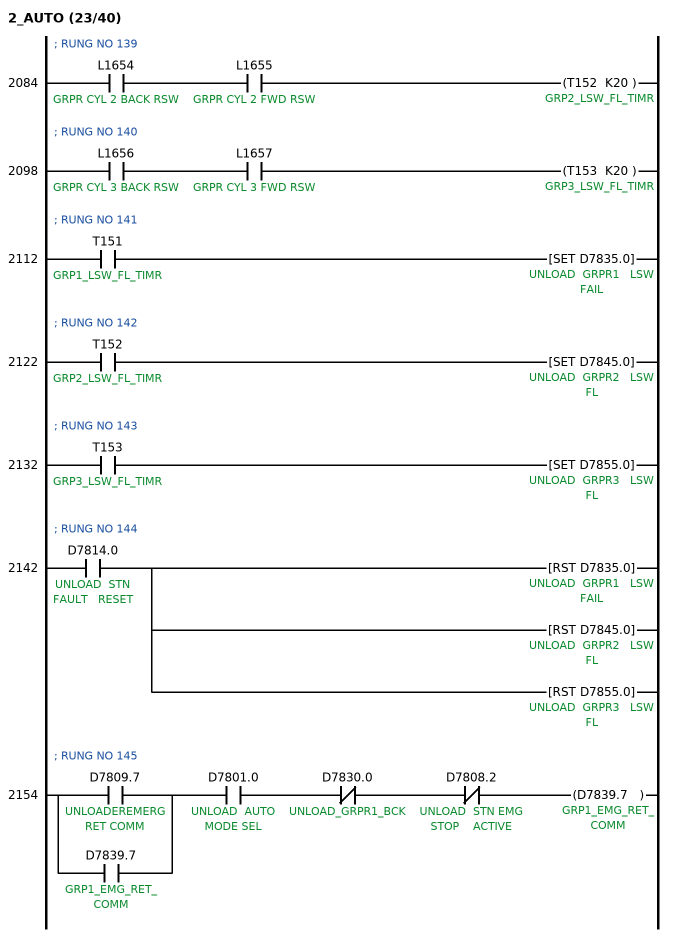
; RUNG NO 139
2084  LD      L1654  ; GRPR CYL 2 BACK RSW
      AND     L1655  ; GRPR CYL 2 FWD RSW
      OUT     T152 K20  ; GRP2_LSW_FL_TIMR
; RUNG NO 140
2098  LD      L1656  ; GRPR CYL 3 BACK RSW
      AND     L1657  ; GRPR CYL 3 FWD RSW
      OUT     T153 K20  ; GRP3_LSW_FL_TIMR
; RUNG NO 141
2112  LD      T151  ; GRP1_LSW_FL_TIMR
      SET     D7835.0  ; UNLOAD  GRPR1   LSW FAIL
; RUNG NO 142
2122  LD      T152  ; GRP2_LSW_FL_TIMR
      SET     D7845.0  ; UNLOAD  GRPR2   LSW FL
; RUNG NO 143
2132  LD      T153  ; GRP3_LSW_FL_TIMR
      SET     D7855.0  ; UNLOAD  GRPR3   LSW FL
; RUNG NO 144
2142  LD      D7814.0  ; UNLOAD  STN     FAULT   RESET
      RST     D7835.0  ; UNLOAD  GRPR1   LSW FAIL
      RST     D7845.0  ; UNLOAD  GRPR2   LSW FL
      RST     D7855.0  ; UNLOAD  GRPR3   LSW FL
; RUNG NO 145
2154  LD      D7809.7  ; UNLOADEREMERG   RET COMM
      OR      D7839.7  ; GRP1_EMG_RET_COMM
      AND     D7801.0  ; UNLOAD  AUTO    MODE SEL
      ANI     D7830.0  ; UNLOAD_GRPR1_BCK
      ANI     D7808.2  ; UNLOAD  STN EMG STOP    ACTIVE
      OUT     D7839.7  ; GRP1_EMG_RET_COMM
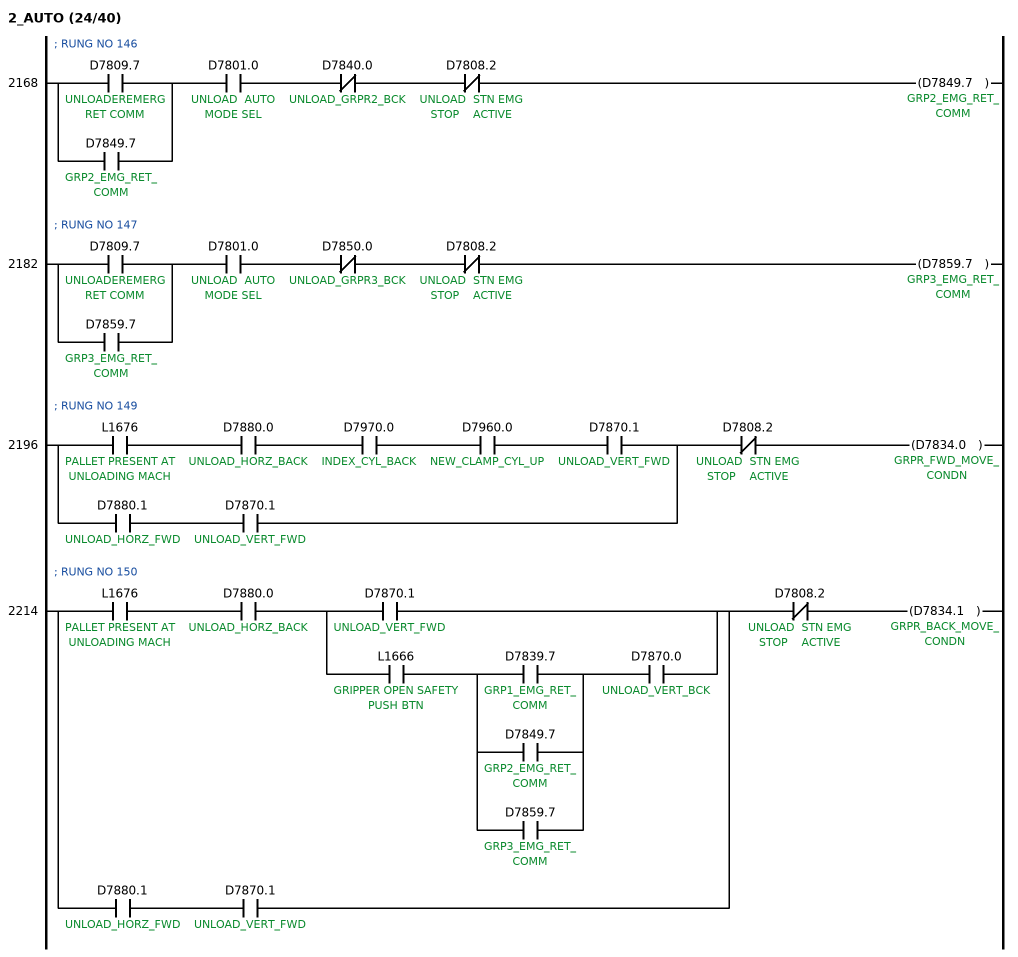
; RUNG NO 146
2168  LD      D7809.7  ; UNLOADEREMERG   RET COMM
      OR      D7849.7  ; GRP2_EMG_RET_COMM
      AND     D7801.0  ; UNLOAD  AUTO    MODE SEL
      ANI     D7840.0  ; UNLOAD_GRPR2_BCK
      ANI     D7808.2  ; UNLOAD  STN EMG STOP    ACTIVE
      OUT     D7849.7  ; GRP2_EMG_RET_COMM
; RUNG NO 147
2182  LD      D7809.7  ; UNLOADEREMERG   RET COMM
      OR      D7859.7  ; GRP3_EMG_RET_COMM
      AND     D7801.0  ; UNLOAD  AUTO    MODE SEL
      ANI     D7850.0  ; UNLOAD_GRPR3_BCK
      ANI     D7808.2  ; UNLOAD  STN EMG STOP    ACTIVE
      OUT     D7859.7  ; GRP3_EMG_RET_COMM
; RUNG NO 149
2196  LD      L1676  ; PALLET PRESENT AT UNLOADING MACH
      AND     D7880.0  ; UNLOAD_HORZ_BACK
      AND     D7970.0  ; INDEX_CYL_BACK
      AND     D7960.0  ; NEW_CLAMP_CYL_UP
      AND     D7870.1  ; UNLOAD_VERT_FWD
      LD      D7880.1  ; UNLOAD_HORZ_FWD
      AND     D7870.1  ; UNLOAD_VERT_FWD
      ORB
      ANI     D7808.2  ; UNLOAD  STN EMG STOP    ACTIVE
      OUT     D7834.0  ; GRPR_FWD_MOVE_CONDN
; RUNG NO 150
2214  LD      L1676  ; PALLET PRESENT AT UNLOADING MACH
      AND     D7880.0  ; UNLOAD_HORZ_BACK
      LD      D7870.1  ; UNLOAD_VERT_FWD
      LD      L1666  ; GRIPPER OPEN SAFETY PUSH BTN
      LD      D7839.7  ; GRP1_EMG_RET_COMM
      OR      D7849.7  ; GRP2_EMG_RET_COMM
      OR      D7859.7  ; GRP3_EMG_RET_COMM
      ANB
      AND     D7870.0  ; UNLOAD_VERT_BCK
      ORB
      ANB
      LD      D7880.1  ; UNLOAD_HORZ_FWD
      AND     D7870.1  ; UNLOAD_VERT_FWD
      ORB
      ANI     D7808.2  ; UNLOAD  STN EMG STOP    ACTIVE
      OUT     D7834.1  ; GRPR_BACK_MOVE_CONDN
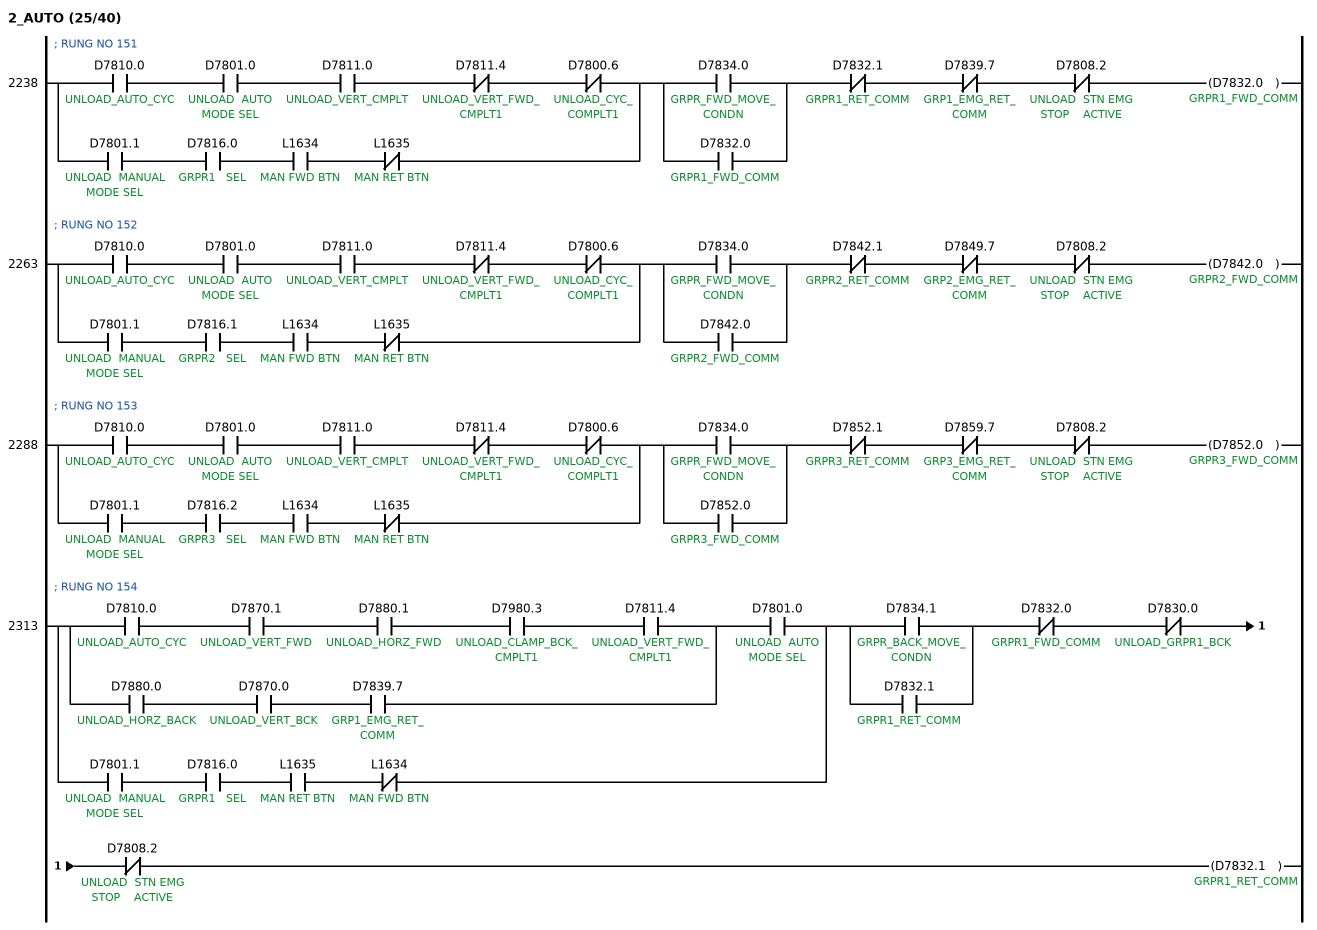
; RUNG NO 151
2238  LD      D7810.0  ; UNLOAD_AUTO_CYC
      AND     D7801.0  ; UNLOAD  AUTO    MODE SEL
      AND     D7811.0  ; UNLOAD_VERT_CMPLT
      ANI     D7811.4  ; UNLOAD_VERT_FWD_CMPLT1
      ANI     D7800.6  ; UNLOAD_CYC_COMPLT1
      LD      D7801.1  ; UNLOAD  MANUAL  MODE SEL
      AND     D7816.0  ; GRPR1   SEL
      AND     L1634  ; MAN FWD BTN
      ANI     L1635  ; MAN RET BTN
      ORB
      LD      D7834.0  ; GRPR_FWD_MOVE_CONDN
      OR      D7832.0  ; GRPR1_FWD_COMM
      ANB
      ANI     D7832.1  ; GRPR1_RET_COMM
      ANI     D7839.7  ; GRP1_EMG_RET_COMM
      ANI     D7808.2  ; UNLOAD  STN EMG STOP    ACTIVE
      OUT     D7832.0  ; GRPR1_FWD_COMM
; RUNG NO 152
2263  LD      D7810.0  ; UNLOAD_AUTO_CYC
      AND     D7801.0  ; UNLOAD  AUTO    MODE SEL
      AND     D7811.0  ; UNLOAD_VERT_CMPLT
      ANI     D7811.4  ; UNLOAD_VERT_FWD_CMPLT1
      ANI     D7800.6  ; UNLOAD_CYC_COMPLT1
      LD      D7801.1  ; UNLOAD  MANUAL  MODE SEL
      AND     D7816.1  ; GRPR2   SEL
      AND     L1634  ; MAN FWD BTN
      ANI     L1635  ; MAN RET BTN
      ORB
      LD      D7834.0  ; GRPR_FWD_MOVE_CONDN
      OR      D7842.0  ; GRPR2_FWD_COMM
      ANB
      ANI     D7842.1  ; GRPR2_RET_COMM
      ANI     D7849.7  ; GRP2_EMG_RET_COMM
      ANI     D7808.2  ; UNLOAD  STN EMG STOP    ACTIVE
      OUT     D7842.0  ; GRPR2_FWD_COMM
; RUNG NO 153
2288  LD      D7810.0  ; UNLOAD_AUTO_CYC
      AND     D7801.0  ; UNLOAD  AUTO    MODE SEL
      AND     D7811.0  ; UNLOAD_VERT_CMPLT
      ANI     D7811.4  ; UNLOAD_VERT_FWD_CMPLT1
      ANI     D7800.6  ; UNLOAD_CYC_COMPLT1
      LD      D7801.1  ; UNLOAD  MANUAL  MODE SEL
      AND     D7816.2  ; GRPR3   SEL
      AND     L1634  ; MAN FWD BTN
      ANI     L1635  ; MAN RET BTN
      ORB
      LD      D7834.0  ; GRPR_FWD_MOVE_CONDN
      OR      D7852.0  ; GRPR3_FWD_COMM
      ANB
      ANI     D7852.1  ; GRPR3_RET_COMM
      ANI     D7859.7  ; GRP3_EMG_RET_COMM
      ANI     D7808.2  ; UNLOAD  STN EMG STOP    ACTIVE
      OUT     D7852.0  ; GRPR3_FWD_COMM
; RUNG NO 154
2313  LD      D7810.0  ; UNLOAD_AUTO_CYC
      AND     D7870.1  ; UNLOAD_VERT_FWD
      AND     D7880.1  ; UNLOAD_HORZ_FWD
      AND     D7980.3  ; UNLOAD_CLAMP_BCK_CMPLT1
      AND     D7811.4  ; UNLOAD_VERT_FWD_CMPLT1
      LD      D7880.0  ; UNLOAD_HORZ_BACK
      AND     D7870.0  ; UNLOAD_VERT_BCK
      AND     D7839.7  ; GRP1_EMG_RET_COMM
      ORB
      AND     D7801.0  ; UNLOAD  AUTO    MODE SEL
      LD      D7801.1  ; UNLOAD  MANUAL  MODE SEL
      AND     D7816.0  ; GRPR1   SEL
      AND     L1635  ; MAN RET BTN
      ANI     L1634  ; MAN FWD BTN
      ORB
      LD      D7834.1  ; GRPR_BACK_MOVE_CONDN
      OR      D7832.1  ; GRPR1_RET_COMM
      ANB
      ANI     D7832.0  ; GRPR1_FWD_COMM
      ANI     D7830.0  ; UNLOAD_GRPR1_BCK
      ANI     D7808.2  ; UNLOAD  STN EMG STOP    ACTIVE
      OUT     D7832.1  ; GRPR1_RET_COMM
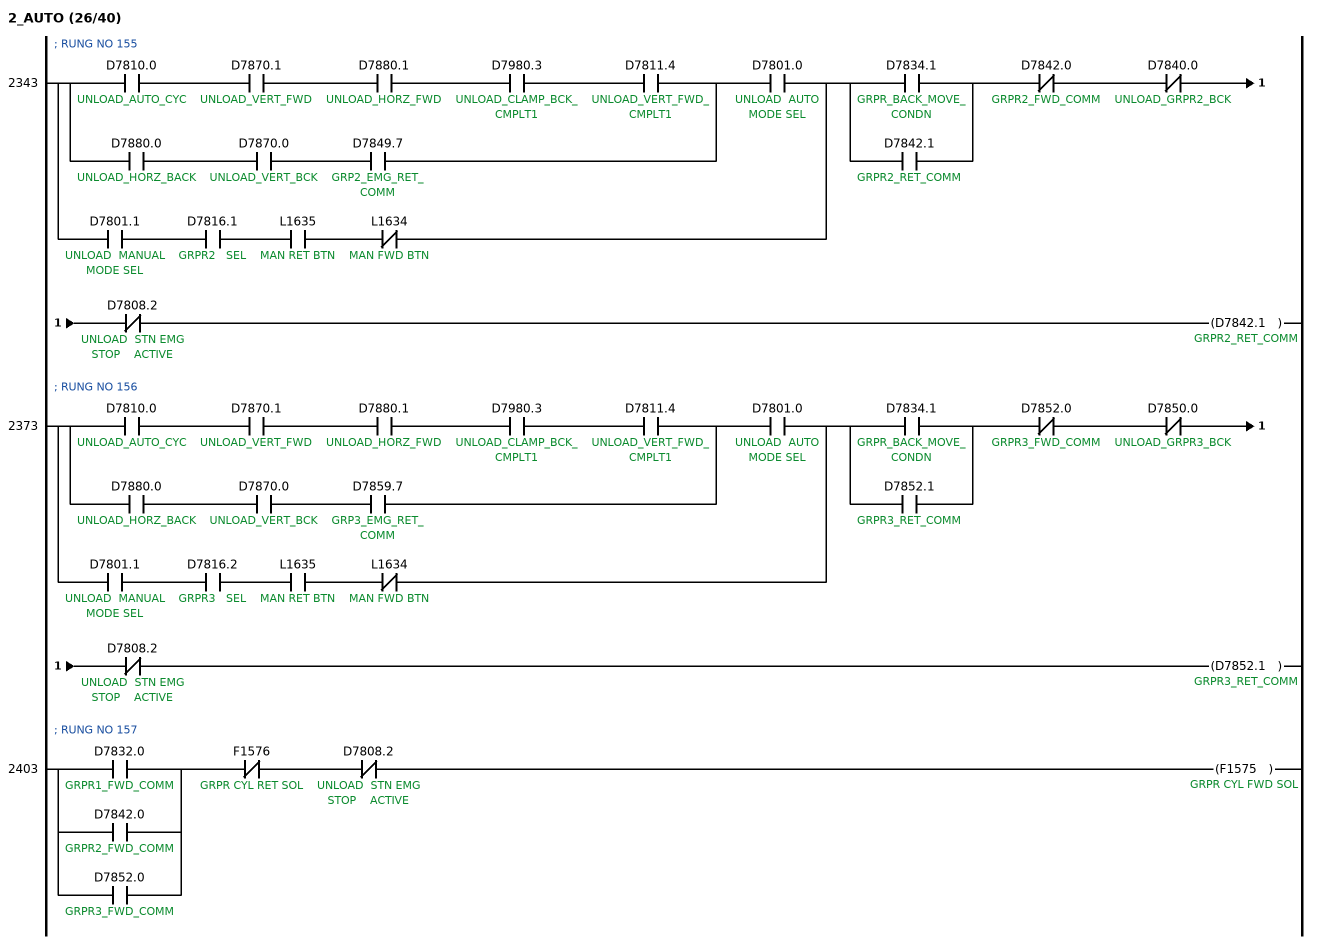
; RUNG NO 155
2343  LD      D7810.0  ; UNLOAD_AUTO_CYC
      AND     D7870.1  ; UNLOAD_VERT_FWD
      AND     D7880.1  ; UNLOAD_HORZ_FWD
      AND     D7980.3  ; UNLOAD_CLAMP_BCK_CMPLT1
      AND     D7811.4  ; UNLOAD_VERT_FWD_CMPLT1
      LD      D7880.0  ; UNLOAD_HORZ_BACK
      AND     D7870.0  ; UNLOAD_VERT_BCK
      AND     D7849.7  ; GRP2_EMG_RET_COMM
      ORB
      AND     D7801.0  ; UNLOAD  AUTO    MODE SEL
      LD      D7801.1  ; UNLOAD  MANUAL  MODE SEL
      AND     D7816.1  ; GRPR2   SEL
      AND     L1635  ; MAN RET BTN
      ANI     L1634  ; MAN FWD BTN
      ORB
      LD      D7834.1  ; GRPR_BACK_MOVE_CONDN
      OR      D7842.1  ; GRPR2_RET_COMM
      ANB
      ANI     D7842.0  ; GRPR2_FWD_COMM
      ANI     D7840.0  ; UNLOAD_GRPR2_BCK
      ANI     D7808.2  ; UNLOAD  STN EMG STOP    ACTIVE
      OUT     D7842.1  ; GRPR2_RET_COMM
; RUNG NO 156
2373  LD      D7810.0  ; UNLOAD_AUTO_CYC
      AND     D7870.1  ; UNLOAD_VERT_FWD
      AND     D7880.1  ; UNLOAD_HORZ_FWD
      AND     D7980.3  ; UNLOAD_CLAMP_BCK_CMPLT1
      AND     D7811.4  ; UNLOAD_VERT_FWD_CMPLT1
      LD      D7880.0  ; UNLOAD_HORZ_BACK
      AND     D7870.0  ; UNLOAD_VERT_BCK
      AND     D7859.7  ; GRP3_EMG_RET_COMM
      ORB
      AND     D7801.0  ; UNLOAD  AUTO    MODE SEL
      LD      D7801.1  ; UNLOAD  MANUAL  MODE SEL
      AND     D7816.2  ; GRPR3   SEL
      AND     L1635  ; MAN RET BTN
      ANI     L1634  ; MAN FWD BTN
      ORB
      LD      D7834.1  ; GRPR_BACK_MOVE_CONDN
      OR      D7852.1  ; GRPR3_RET_COMM
      ANB
      ANI     D7852.0  ; GRPR3_FWD_COMM
      ANI     D7850.0  ; UNLOAD_GRPR3_BCK
      ANI     D7808.2  ; UNLOAD  STN EMG STOP    ACTIVE
      OUT     D7852.1  ; GRPR3_RET_COMM
; RUNG NO 157
2403  LD      D7832.0  ; GRPR1_FWD_COMM
      OR      D7842.0  ; GRPR2_FWD_COMM
      OR      D7852.0  ; GRPR3_FWD_COMM
      ANI     F1576  ; GRPR CYL RET SOL
      ANI     D7808.2  ; UNLOAD  STN EMG STOP    ACTIVE
      OUT     F1575  ; GRPR CYL FWD SOL
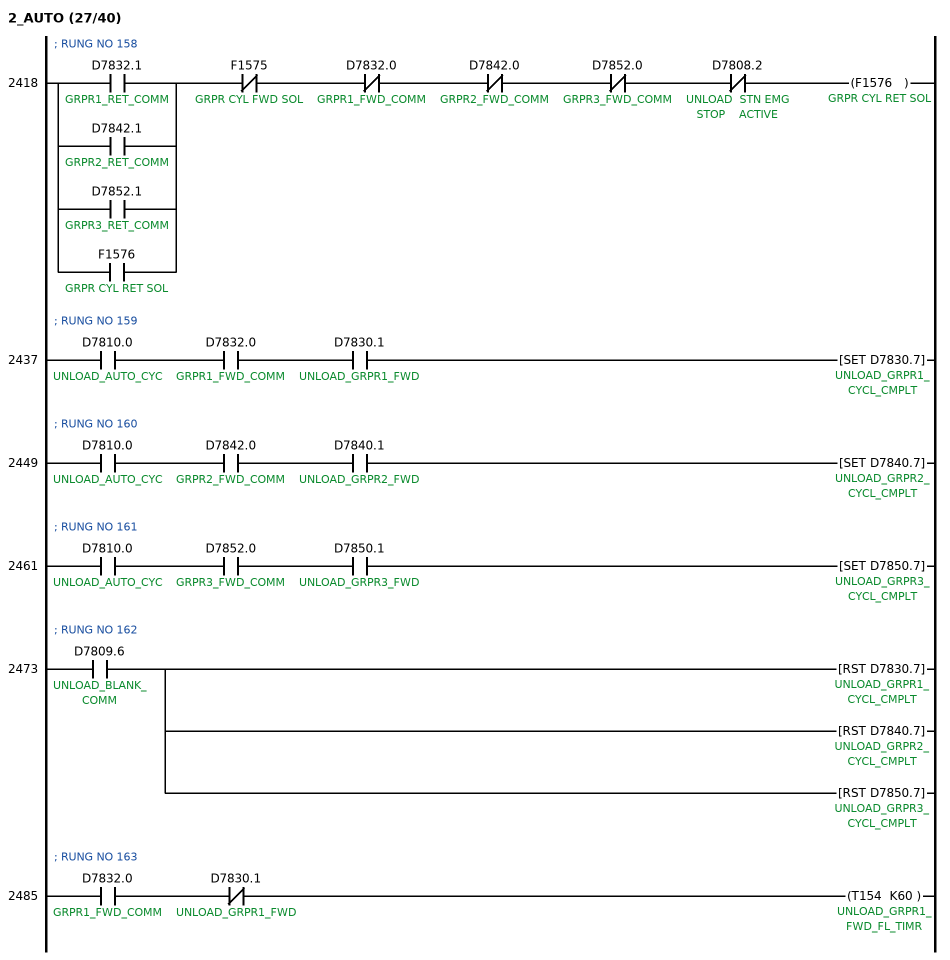
; RUNG NO 158
2418  LD      D7832.1  ; GRPR1_RET_COMM
      OR      D7842.1  ; GRPR2_RET_COMM
      OR      D7852.1  ; GRPR3_RET_COMM
      OR      F1576  ; GRPR CYL RET SOL
      ANI     F1575  ; GRPR CYL FWD SOL
      ANI     D7832.0  ; GRPR1_FWD_COMM
      ANI     D7842.0  ; GRPR2_FWD_COMM
      ANI     D7852.0  ; GRPR3_FWD_COMM
      ANI     D7808.2  ; UNLOAD  STN EMG STOP    ACTIVE
      OUT     F1576  ; GRPR CYL RET SOL
; RUNG NO 159
2437  LD      D7810.0  ; UNLOAD_AUTO_CYC
      AND     D7832.0  ; GRPR1_FWD_COMM
      AND     D7830.1  ; UNLOAD_GRPR1_FWD
      SET     D7830.7  ; UNLOAD_GRPR1_CYCL_CMPLT
; RUNG NO 160
2449  LD      D7810.0  ; UNLOAD_AUTO_CYC
      AND     D7842.0  ; GRPR2_FWD_COMM
      AND     D7840.1  ; UNLOAD_GRPR2_FWD
      SET     D7840.7  ; UNLOAD_GRPR2_CYCL_CMPLT
; RUNG NO 161
2461  LD      D7810.0  ; UNLOAD_AUTO_CYC
      AND     D7852.0  ; GRPR3_FWD_COMM
      AND     D7850.1  ; UNLOAD_GRPR3_FWD
      SET     D7850.7  ; UNLOAD_GRPR3_CYCL_CMPLT
; RUNG NO 162
2473  LD      D7809.6  ; UNLOAD_BLANK_COMM
      RST     D7830.7  ; UNLOAD_GRPR1_CYCL_CMPLT
      RST     D7840.7  ; UNLOAD_GRPR2_CYCL_CMPLT
      RST     D7850.7  ; UNLOAD_GRPR3_CYCL_CMPLT
; RUNG NO 163
2485  LD      D7832.0  ; GRPR1_FWD_COMM
      ANI     D7830.1  ; UNLOAD_GRPR1_FWD
      OUT     T154 K60  ; UNLOAD_GRPR1_FWD_FL_TIMR
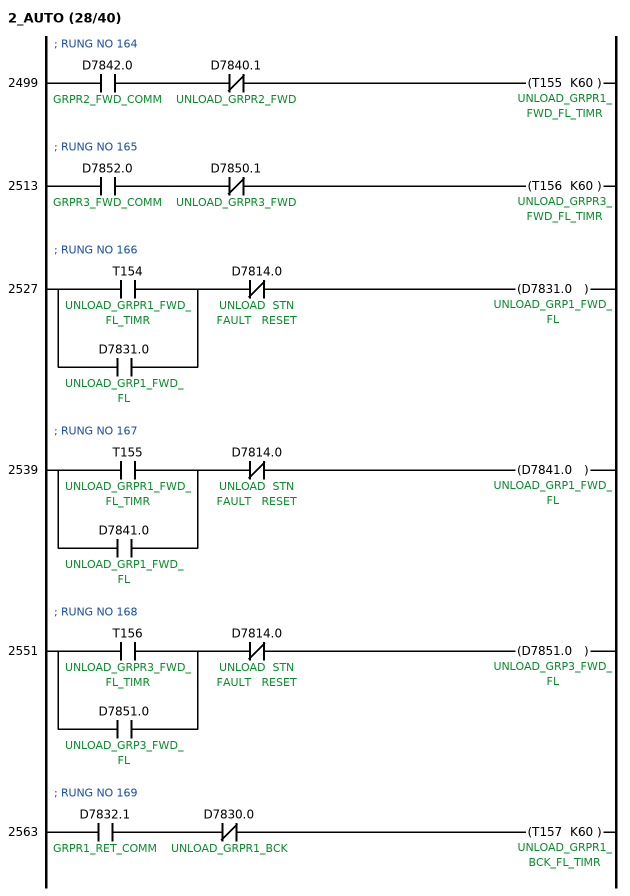
; RUNG NO 164
2499  LD      D7842.0  ; GRPR2_FWD_COMM
      ANI     D7840.1  ; UNLOAD_GRPR2_FWD
      OUT     T155 K60  ; UNLOAD_GRPR1_FWD_FL_TIMR
; RUNG NO 165
2513  LD      D7852.0  ; GRPR3_FWD_COMM
      ANI     D7850.1  ; UNLOAD_GRPR3_FWD
      OUT     T156 K60  ; UNLOAD_GRPR3_FWD_FL_TIMR
; RUNG NO 166
2527  LD      T154  ; UNLOAD_GRPR1_FWD_FL_TIMR
      OR      D7831.0  ; UNLOAD_GRP1_FWD_FL
      ANI     D7814.0  ; UNLOAD  STN     FAULT   RESET
      OUT     D7831.0  ; UNLOAD_GRP1_FWD_FL
; RUNG NO 167
2539  LD      T155  ; UNLOAD_GRPR1_FWD_FL_TIMR
      OR      D7841.0  ; UNLOAD_GRP1_FWD_FL
      ANI     D7814.0  ; UNLOAD  STN     FAULT   RESET
      OUT     D7841.0  ; UNLOAD_GRP1_FWD_FL
; RUNG NO 168
2551  LD      T156  ; UNLOAD_GRPR3_FWD_FL_TIMR
      OR      D7851.0  ; UNLOAD_GRP3_FWD_FL
      ANI     D7814.0  ; UNLOAD  STN     FAULT   RESET
      OUT     D7851.0  ; UNLOAD_GRP3_FWD_FL
; RUNG NO 169
2563  LD      D7832.1  ; GRPR1_RET_COMM
      ANI     D7830.0  ; UNLOAD_GRPR1_BCK
      OUT     T157 K60  ; UNLOAD_GRPR1_BCK_FL_TIMR
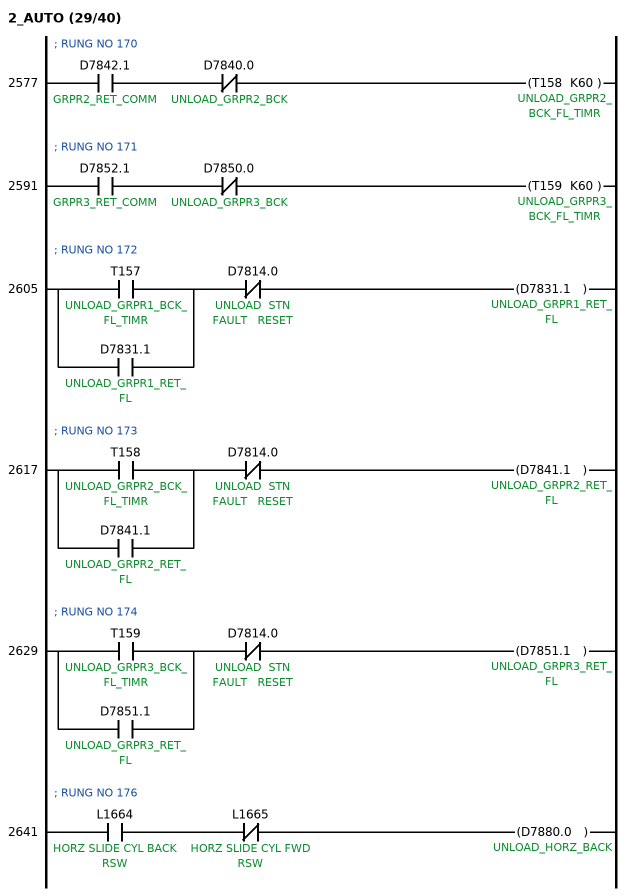
; RUNG NO 170
2577  LD      D7842.1  ; GRPR2_RET_COMM
      ANI     D7840.0  ; UNLOAD_GRPR2_BCK
      OUT     T158 K60  ; UNLOAD_GRPR2_BCK_FL_TIMR
; RUNG NO 171
2591  LD      D7852.1  ; GRPR3_RET_COMM
      ANI     D7850.0  ; UNLOAD_GRPR3_BCK
      OUT     T159 K60  ; UNLOAD_GRPR3_BCK_FL_TIMR
; RUNG NO 172
2605  LD      T157  ; UNLOAD_GRPR1_BCK_FL_TIMR
      OR      D7831.1  ; UNLOAD_GRPR1_RET_FL
      ANI     D7814.0  ; UNLOAD  STN     FAULT   RESET
      OUT     D7831.1  ; UNLOAD_GRPR1_RET_FL
; RUNG NO 173
2617  LD      T158  ; UNLOAD_GRPR2_BCK_FL_TIMR
      OR      D7841.1  ; UNLOAD_GRPR2_RET_FL
      ANI     D7814.0  ; UNLOAD  STN     FAULT   RESET
      OUT     D7841.1  ; UNLOAD_GRPR2_RET_FL
; RUNG NO 174
2629  LD      T159  ; UNLOAD_GRPR3_BCK_FL_TIMR
      OR      D7851.1  ; UNLOAD_GRPR3_RET_FL
      ANI     D7814.0  ; UNLOAD  STN     FAULT   RESET
      OUT     D7851.1  ; UNLOAD_GRPR3_RET_FL
; RUNG NO 176
2641  LD      L1664  ; HORZ SLIDE CYL BACK RSW
      ANI     L1665  ; HORZ SLIDE CYL FWD RSW
      OUT     D7880.0  ; UNLOAD_HORZ_BACK
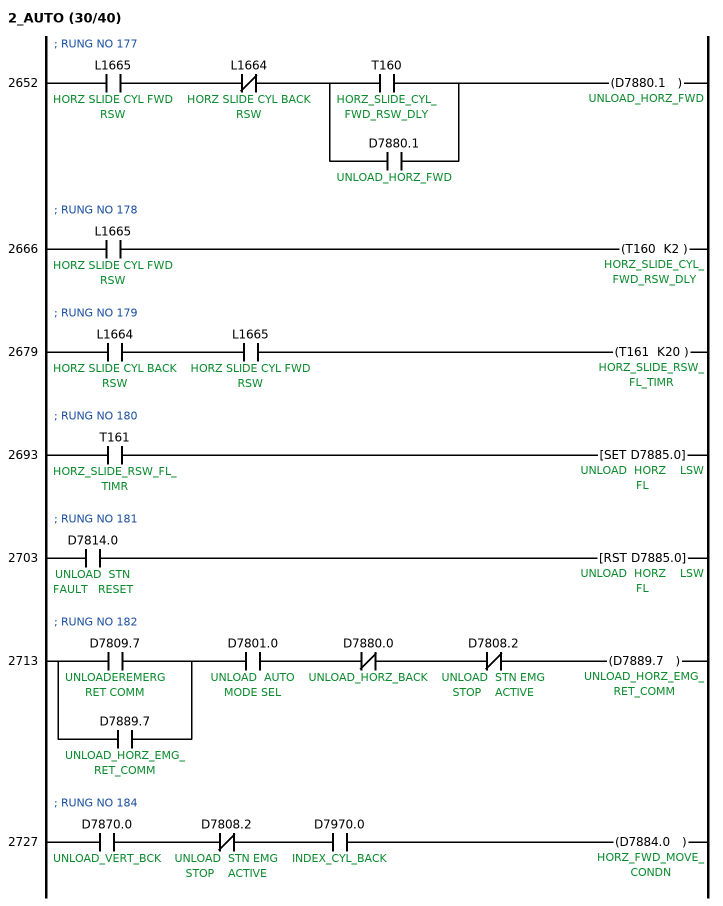
; RUNG NO 177
2652  LD      L1665  ; HORZ SLIDE CYL FWD RSW
      ANI     L1664  ; HORZ SLIDE CYL BACK RSW
      LD      T160  ; HORZ_SLIDE_CYL_FWD_RSW_DLY
      OR      D7880.1  ; UNLOAD_HORZ_FWD
      ANB
      OUT     D7880.1  ; UNLOAD_HORZ_FWD
; RUNG NO 178
2666  LD      L1665  ; HORZ SLIDE CYL FWD RSW
      OUT     T160 K2  ; HORZ_SLIDE_CYL_FWD_RSW_DLY
; RUNG NO 179
2679  LD      L1664  ; HORZ SLIDE CYL BACK RSW
      AND     L1665  ; HORZ SLIDE CYL FWD RSW
      OUT     T161 K20  ; HORZ_SLIDE_RSW_FL_TIMR
; RUNG NO 180
2693  LD      T161  ; HORZ_SLIDE_RSW_FL_TIMR
      SET     D7885.0  ; UNLOAD  HORZ    LSW FL
; RUNG NO 181
2703  LD      D7814.0  ; UNLOAD  STN     FAULT   RESET
      RST     D7885.0  ; UNLOAD  HORZ    LSW FL
; RUNG NO 182
2713  LD      D7809.7  ; UNLOADEREMERG   RET COMM
      OR      D7889.7  ; UNLOAD_HORZ_EMG_RET_COMM
      AND     D7801.0  ; UNLOAD  AUTO    MODE SEL
      ANI     D7880.0  ; UNLOAD_HORZ_BACK
      ANI     D7808.2  ; UNLOAD  STN EMG STOP    ACTIVE
      OUT     D7889.7  ; UNLOAD_HORZ_EMG_RET_COMM
; RUNG NO 184
2727  LD      D7870.0  ; UNLOAD_VERT_BCK
      ANI     D7808.2  ; UNLOAD  STN EMG STOP    ACTIVE
      AND     D7970.0  ; INDEX_CYL_BACK
      OUT     D7884.0  ; HORZ_FWD_MOVE_CONDN
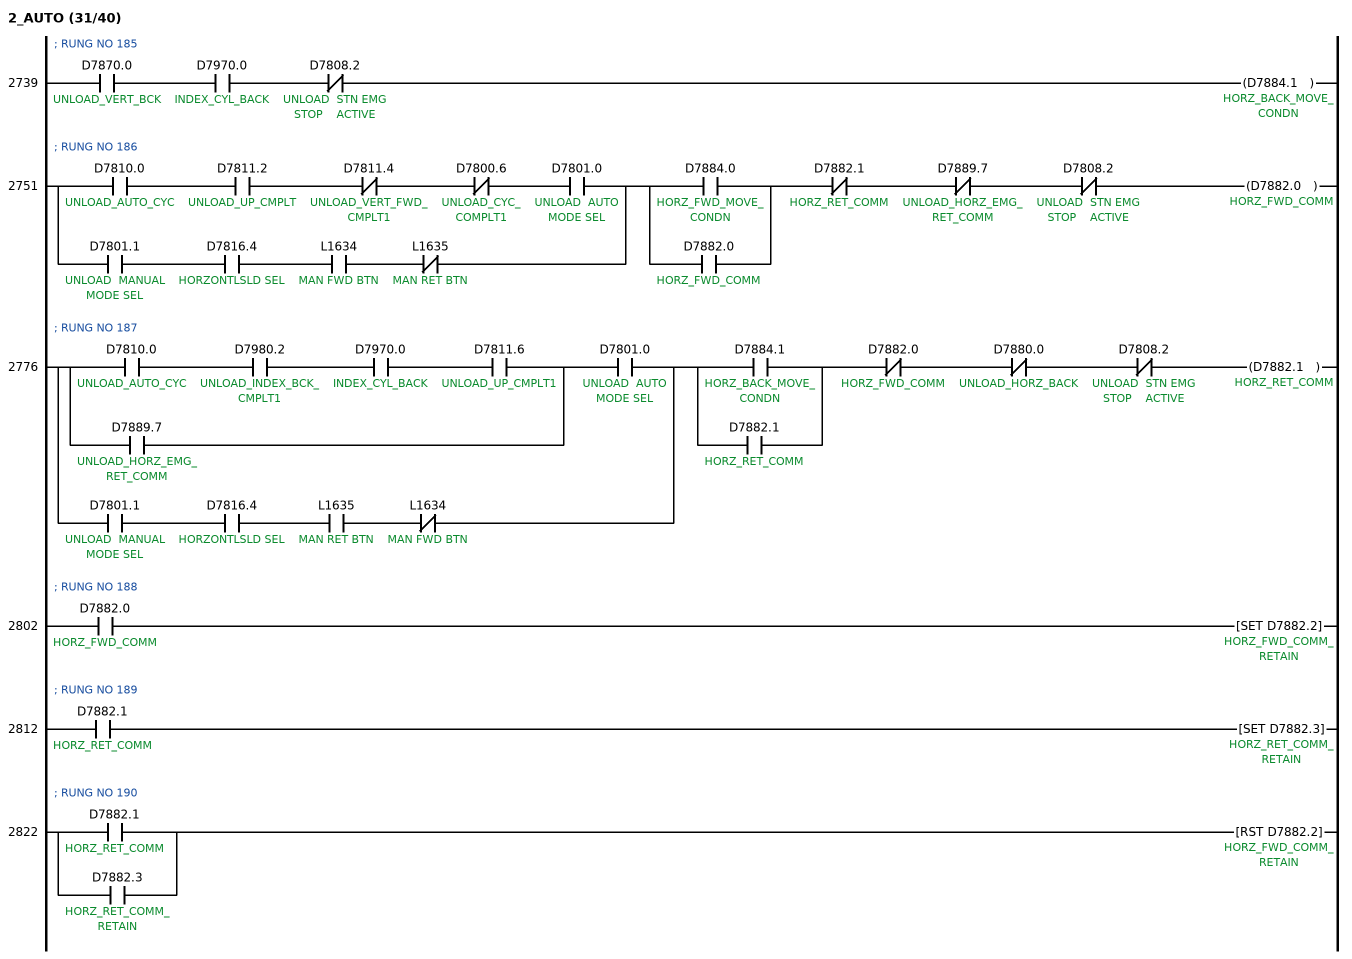
; RUNG NO 185
2739  LD      D7870.0  ; UNLOAD_VERT_BCK
      AND     D7970.0  ; INDEX_CYL_BACK
      ANI     D7808.2  ; UNLOAD  STN EMG STOP    ACTIVE
      OUT     D7884.1  ; HORZ_BACK_MOVE_CONDN
; RUNG NO 186
2751  LD      D7810.0  ; UNLOAD_AUTO_CYC
      AND     D7811.2  ; UNLOAD_UP_CMPLT
      ANI     D7811.4  ; UNLOAD_VERT_FWD_CMPLT1
      ANI     D7800.6  ; UNLOAD_CYC_COMPLT1
      AND     D7801.0  ; UNLOAD  AUTO    MODE SEL
      LD      D7801.1  ; UNLOAD  MANUAL  MODE SEL
      AND     D7816.4  ; HORZONTLSLD SEL
      AND     L1634  ; MAN FWD BTN
      ANI     L1635  ; MAN RET BTN
      ORB
      LD      D7884.0  ; HORZ_FWD_MOVE_CONDN
      OR      D7882.0  ; HORZ_FWD_COMM
      ANB
      ANI     D7882.1  ; HORZ_RET_COMM
      ANI     D7889.7  ; UNLOAD_HORZ_EMG_RET_COMM
      ANI     D7808.2  ; UNLOAD  STN EMG STOP    ACTIVE
      OUT     D7882.0  ; HORZ_FWD_COMM
; RUNG NO 187
2776  LD      D7810.0  ; UNLOAD_AUTO_CYC
      AND     D7980.2  ; UNLOAD_INDEX_BCK_CMPLT1
      AND     D7970.0  ; INDEX_CYL_BACK
      AND     D7811.6  ; UNLOAD_UP_CMPLT1
      OR      D7889.7  ; UNLOAD_HORZ_EMG_RET_COMM
      AND     D7801.0  ; UNLOAD  AUTO    MODE SEL
      LD      D7801.1  ; UNLOAD  MANUAL  MODE SEL
      AND     D7816.4  ; HORZONTLSLD SEL
      AND     L1635  ; MAN RET BTN
      ANI     L1634  ; MAN FWD BTN
      ORB
      LD      D7884.1  ; HORZ_BACK_MOVE_CONDN
      OR      D7882.1  ; HORZ_RET_COMM
      ANB
      ANI     D7882.0  ; HORZ_FWD_COMM
      ANI     D7880.0  ; UNLOAD_HORZ_BACK
      ANI     D7808.2  ; UNLOAD  STN EMG STOP    ACTIVE
      OUT     D7882.1  ; HORZ_RET_COMM
; RUNG NO 188
2802  LD      D7882.0  ; HORZ_FWD_COMM
      SET     D7882.2  ; HORZ_FWD_COMM_RETAIN
; RUNG NO 189
2812  LD      D7882.1  ; HORZ_RET_COMM
      SET     D7882.3  ; HORZ_RET_COMM_RETAIN
; RUNG NO 190
2822  LD      D7882.1  ; HORZ_RET_COMM
      OR      D7882.3  ; HORZ_RET_COMM_RETAIN
      RST     D7882.2  ; HORZ_FWD_COMM_RETAIN
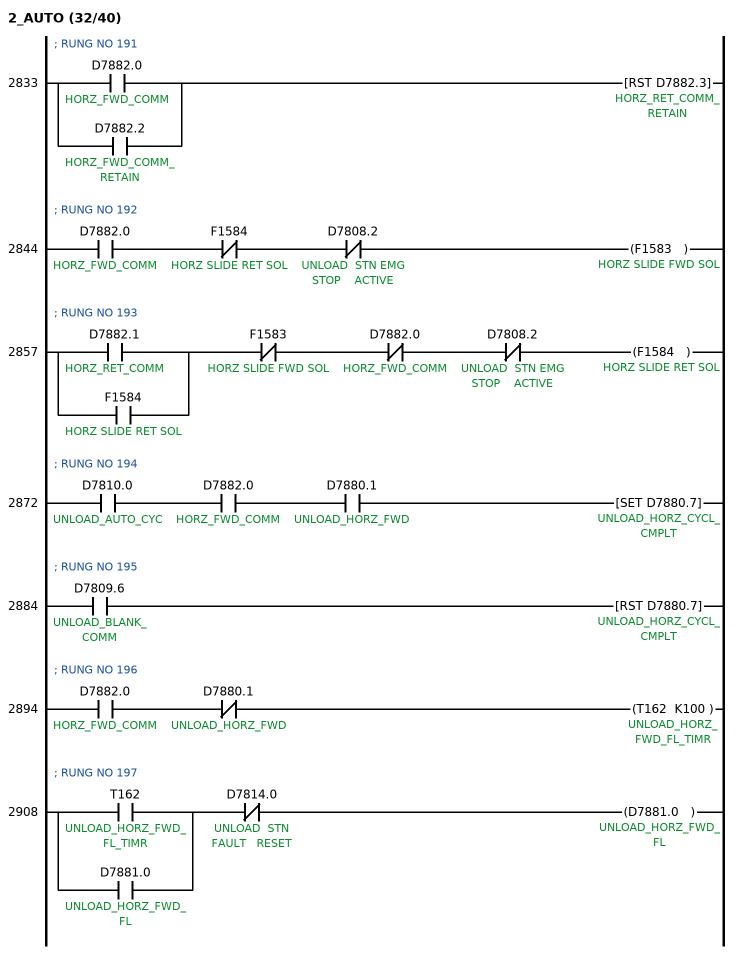
; RUNG NO 191
2833  LD      D7882.0  ; HORZ_FWD_COMM
      OR      D7882.2  ; HORZ_FWD_COMM_RETAIN
      RST     D7882.3  ; HORZ_RET_COMM_RETAIN
; RUNG NO 192
2844  LD      D7882.0  ; HORZ_FWD_COMM
      ANI     F1584  ; HORZ SLIDE RET SOL
      ANI     D7808.2  ; UNLOAD  STN EMG STOP    ACTIVE
      OUT     F1583  ; HORZ SLIDE FWD SOL
; RUNG NO 193
2857  LD      D7882.1  ; HORZ_RET_COMM
      OR      F1584  ; HORZ SLIDE RET SOL
      ANI     F1583  ; HORZ SLIDE FWD SOL
      ANI     D7882.0  ; HORZ_FWD_COMM
      ANI     D7808.2  ; UNLOAD  STN EMG STOP    ACTIVE
      OUT     F1584  ; HORZ SLIDE RET SOL
; RUNG NO 194
2872  LD      D7810.0  ; UNLOAD_AUTO_CYC
      AND     D7882.0  ; HORZ_FWD_COMM
      AND     D7880.1  ; UNLOAD_HORZ_FWD
      SET     D7880.7  ; UNLOAD_HORZ_CYCL_CMPLT
; RUNG NO 195
2884  LD      D7809.6  ; UNLOAD_BLANK_COMM
      RST     D7880.7  ; UNLOAD_HORZ_CYCL_CMPLT
; RUNG NO 196
2894  LD      D7882.0  ; HORZ_FWD_COMM
      ANI     D7880.1  ; UNLOAD_HORZ_FWD
      OUT     T162 K100  ; UNLOAD_HORZ_FWD_FL_TIMR
; RUNG NO 197
2908  LD      T162  ; UNLOAD_HORZ_FWD_FL_TIMR
      OR      D7881.0  ; UNLOAD_HORZ_FWD_FL
      ANI     D7814.0  ; UNLOAD  STN     FAULT   RESET
      OUT     D7881.0  ; UNLOAD_HORZ_FWD_FL
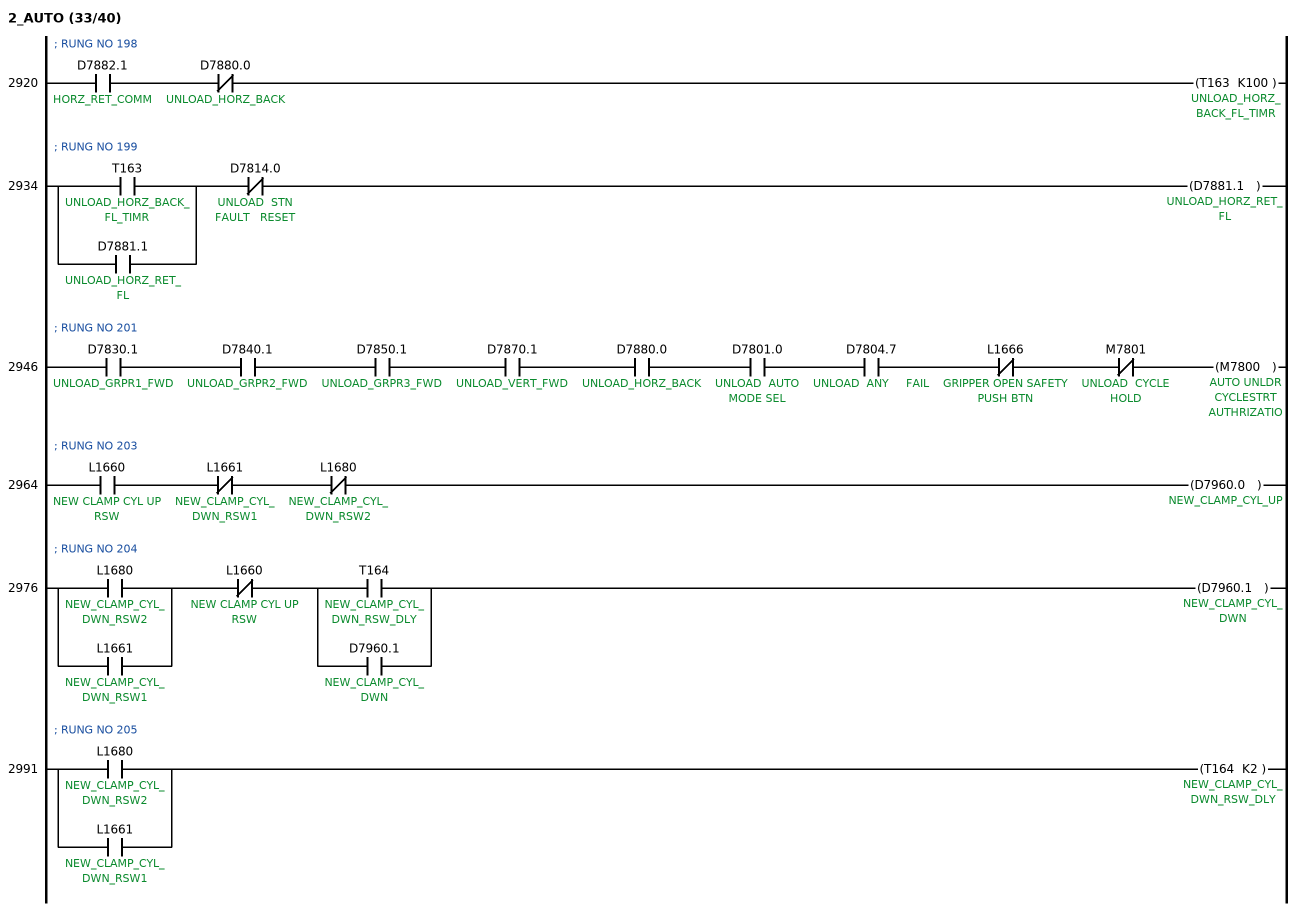
; RUNG NO 198
2920  LD      D7882.1  ; HORZ_RET_COMM
      ANI     D7880.0  ; UNLOAD_HORZ_BACK
      OUT     T163 K100  ; UNLOAD_HORZ_BACK_FL_TIMR
; RUNG NO 199
2934  LD      T163  ; UNLOAD_HORZ_BACK_FL_TIMR
      OR      D7881.1  ; UNLOAD_HORZ_RET_FL
      ANI     D7814.0  ; UNLOAD  STN     FAULT   RESET
      OUT     D7881.1  ; UNLOAD_HORZ_RET_FL
; RUNG NO 201
2946  LD      D7830.1  ; UNLOAD_GRPR1_FWD
      AND     D7840.1  ; UNLOAD_GRPR2_FWD
      AND     D7850.1  ; UNLOAD_GRPR3_FWD
      AND     D7870.1  ; UNLOAD_VERT_FWD
      AND     D7880.0  ; UNLOAD_HORZ_BACK
      AND     D7801.0  ; UNLOAD  AUTO    MODE SEL
      AND     D7804.7  ; UNLOAD  ANY     FAIL
      ANI     L1666  ; GRIPPER OPEN SAFETY PUSH BTN
      ANI     M7801  ; UNLOAD  CYCLE   HOLD
      OUT     M7800  ; AUTO UNLDR CYCLESTRT AUTHRIZATIO
; RUNG NO 203
2964  LD      L1660  ; NEW CLAMP CYL UP RSW
      ANI     L1661  ; NEW_CLAMP_CYL_DWN_RSW1
      ANI     L1680  ; NEW_CLAMP_CYL_DWN_RSW2
      OUT     D7960.0  ; NEW_CLAMP_CYL_UP
; RUNG NO 204
2976  LD      L1680  ; NEW_CLAMP_CYL_DWN_RSW2
      OR      L1661  ; NEW_CLAMP_CYL_DWN_RSW1
      ANI     L1660  ; NEW CLAMP CYL UP RSW
      LD      T164  ; NEW_CLAMP_CYL_DWN_RSW_DLY
      OR      D7960.1  ; NEW_CLAMP_CYL_DWN
      ANB
      OUT     D7960.1  ; NEW_CLAMP_CYL_DWN
; RUNG NO 205
2991  LD      L1680  ; NEW_CLAMP_CYL_DWN_RSW2
      OR      L1661  ; NEW_CLAMP_CYL_DWN_RSW1
      OUT     T164 K2  ; NEW_CLAMP_CYL_DWN_RSW_DLY
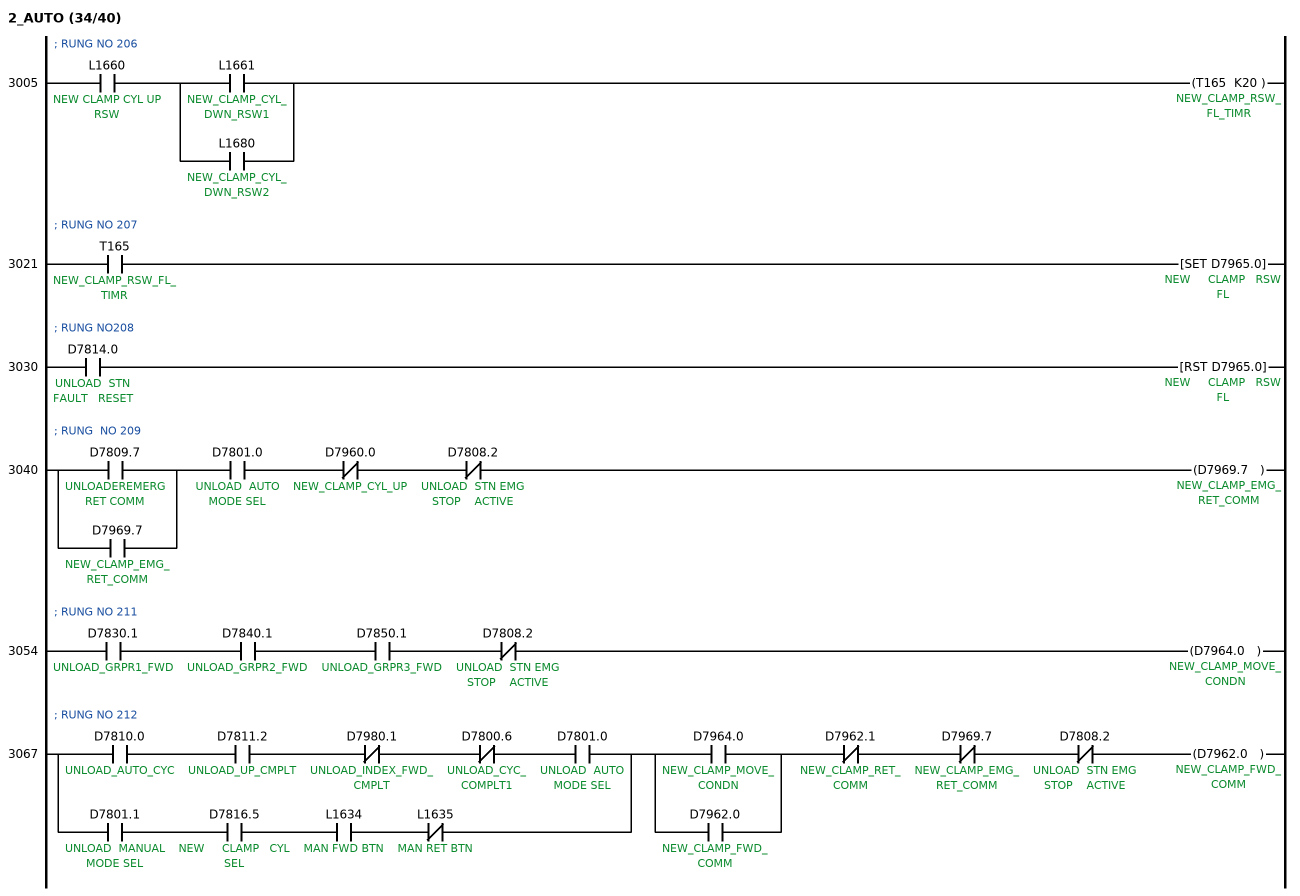
; RUNG NO 206
3005  LD      L1660  ; NEW CLAMP CYL UP RSW
      LD      L1661  ; NEW_CLAMP_CYL_DWN_RSW1
      OR      L1680  ; NEW_CLAMP_CYL_DWN_RSW2
      ANB
      OUT     T165 K20  ; NEW_CLAMP_RSW_FL_TIMR
; RUNG NO 207
3021  LD      T165  ; NEW_CLAMP_RSW_FL_TIMR
      SET     D7965.0  ; NEW     CLAMP   RSW FL
; RUNG NO208
3030  LD      D7814.0  ; UNLOAD  STN     FAULT   RESET
      RST     D7965.0  ; NEW     CLAMP   RSW FL
; RUNG  NO 209
3040  LD      D7809.7  ; UNLOADEREMERG   RET COMM
      OR      D7969.7  ; NEW_CLAMP_EMG_RET_COMM
      AND     D7801.0  ; UNLOAD  AUTO    MODE SEL
      ANI     D7960.0  ; NEW_CLAMP_CYL_UP
      ANI     D7808.2  ; UNLOAD  STN EMG STOP    ACTIVE
      OUT     D7969.7  ; NEW_CLAMP_EMG_RET_COMM
; RUNG NO 211
3054  LD      D7830.1  ; UNLOAD_GRPR1_FWD
      AND     D7840.1  ; UNLOAD_GRPR2_FWD
      AND     D7850.1  ; UNLOAD_GRPR3_FWD
      ANI     D7808.2  ; UNLOAD  STN EMG STOP    ACTIVE
      OUT     D7964.0  ; NEW_CLAMP_MOVE_CONDN
; RUNG NO 212
3067  LD      D7810.0  ; UNLOAD_AUTO_CYC
      AND     D7811.2  ; UNLOAD_UP_CMPLT
      ANI     D7980.1  ; UNLOAD_INDEX_FWD_CMPLT
      ANI     D7800.6  ; UNLOAD_CYC_COMPLT1
      AND     D7801.0  ; UNLOAD  AUTO    MODE SEL
      LD      D7801.1  ; UNLOAD  MANUAL  MODE SEL
      AND     D7816.5  ; NEW     CLAMP   CYL SEL
      AND     L1634  ; MAN FWD BTN
      ANI     L1635  ; MAN RET BTN
      ORB
      LD      D7964.0  ; NEW_CLAMP_MOVE_CONDN
      OR      D7962.0  ; NEW_CLAMP_FWD_COMM
      ANB
      ANI     D7962.1  ; NEW_CLAMP_RET_COMM
      ANI     D7969.7  ; NEW_CLAMP_EMG_RET_COMM
      ANI     D7808.2  ; UNLOAD  STN EMG STOP    ACTIVE
      OUT     D7962.0  ; NEW_CLAMP_FWD_COMM
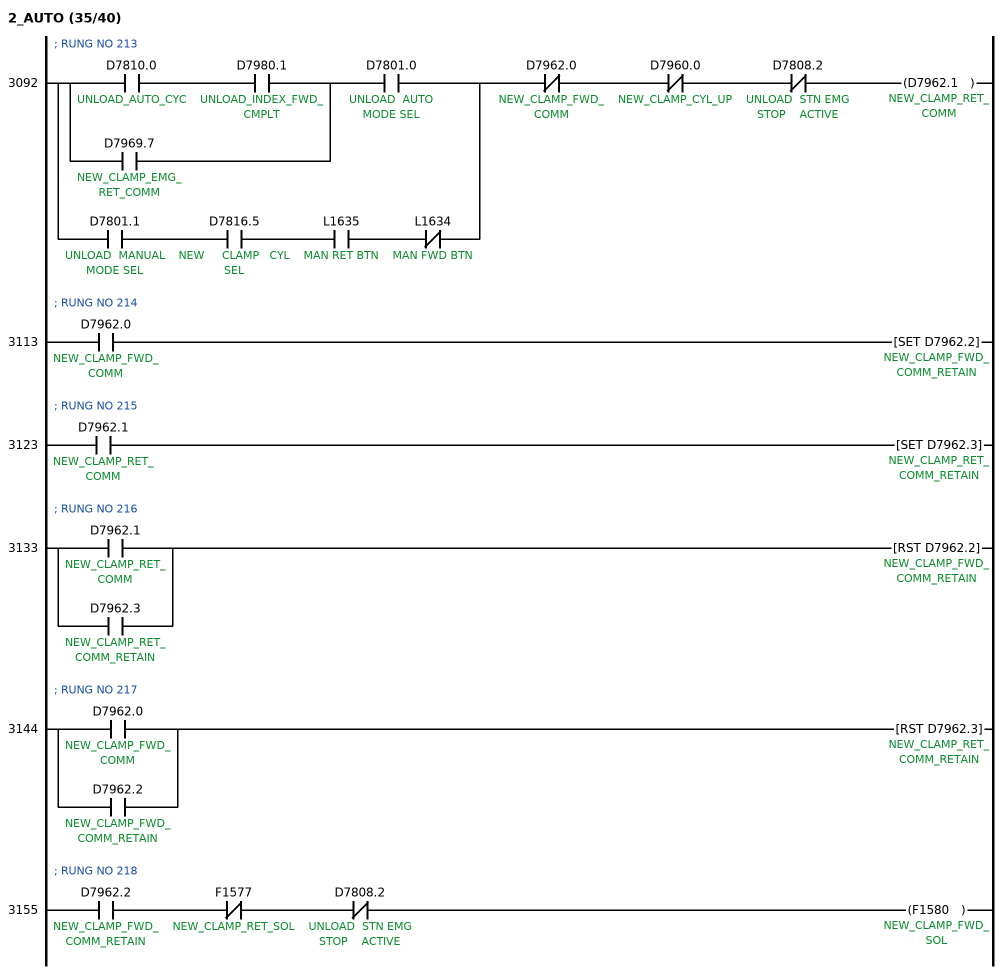
; RUNG NO 213
3092  LD      D7810.0  ; UNLOAD_AUTO_CYC
      AND     D7980.1  ; UNLOAD_INDEX_FWD_CMPLT
      OR      D7969.7  ; NEW_CLAMP_EMG_RET_COMM
      AND     D7801.0  ; UNLOAD  AUTO    MODE SEL
      LD      D7801.1  ; UNLOAD  MANUAL  MODE SEL
      AND     D7816.5  ; NEW     CLAMP   CYL SEL
      AND     L1635  ; MAN RET BTN
      ANI     L1634  ; MAN FWD BTN
      ORB
      ANI     D7962.0  ; NEW_CLAMP_FWD_COMM
      ANI     D7960.0  ; NEW_CLAMP_CYL_UP
      ANI     D7808.2  ; UNLOAD  STN EMG STOP    ACTIVE
      OUT     D7962.1  ; NEW_CLAMP_RET_COMM
; RUNG NO 214
3113  LD      D7962.0  ; NEW_CLAMP_FWD_COMM
      SET     D7962.2  ; NEW_CLAMP_FWD_COMM_RETAIN
; RUNG NO 215
3123  LD      D7962.1  ; NEW_CLAMP_RET_COMM
      SET     D7962.3  ; NEW_CLAMP_RET_COMM_RETAIN
; RUNG NO 216
3133  LD      D7962.1  ; NEW_CLAMP_RET_COMM
      OR      D7962.3  ; NEW_CLAMP_RET_COMM_RETAIN
      RST     D7962.2  ; NEW_CLAMP_FWD_COMM_RETAIN
; RUNG NO 217
3144  LD      D7962.0  ; NEW_CLAMP_FWD_COMM
      OR      D7962.2  ; NEW_CLAMP_FWD_COMM_RETAIN
      RST     D7962.3  ; NEW_CLAMP_RET_COMM_RETAIN
; RUNG NO 218
3155  LD      D7962.2  ; NEW_CLAMP_FWD_COMM_RETAIN
      ANI     F1577  ; NEW_CLAMP_RET_SOL
      ANI     D7808.2  ; UNLOAD  STN EMG STOP    ACTIVE
      OUT     F1580  ; NEW_CLAMP_FWD_SOL
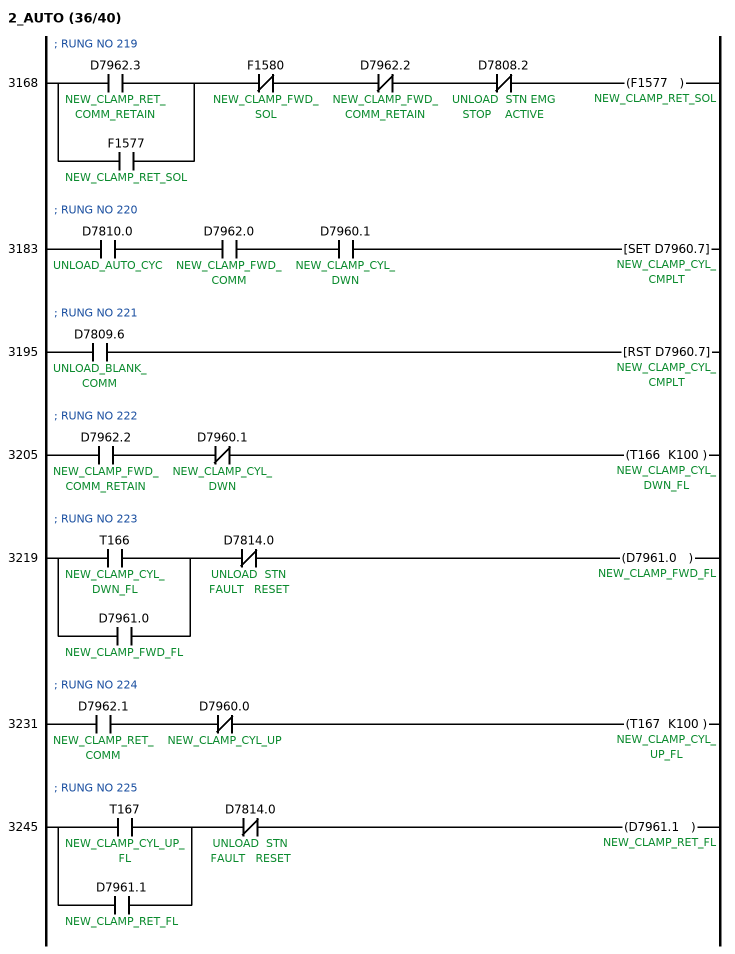
; RUNG NO 219
3168  LD      D7962.3  ; NEW_CLAMP_RET_COMM_RETAIN
      OR      F1577  ; NEW_CLAMP_RET_SOL
      ANI     F1580  ; NEW_CLAMP_FWD_SOL
      ANI     D7962.2  ; NEW_CLAMP_FWD_COMM_RETAIN
      ANI     D7808.2  ; UNLOAD  STN EMG STOP    ACTIVE
      OUT     F1577  ; NEW_CLAMP_RET_SOL
; RUNG NO 220
3183  LD      D7810.0  ; UNLOAD_AUTO_CYC
      AND     D7962.0  ; NEW_CLAMP_FWD_COMM
      AND     D7960.1  ; NEW_CLAMP_CYL_DWN
      SET     D7960.7  ; NEW_CLAMP_CYL_CMPLT
; RUNG NO 221
3195  LD      D7809.6  ; UNLOAD_BLANK_COMM
      RST     D7960.7  ; NEW_CLAMP_CYL_CMPLT
; RUNG NO 222
3205  LD      D7962.2  ; NEW_CLAMP_FWD_COMM_RETAIN
      ANI     D7960.1  ; NEW_CLAMP_CYL_DWN
      OUT     T166 K100  ; NEW_CLAMP_CYL_DWN_FL
; RUNG NO 223
3219  LD      T166  ; NEW_CLAMP_CYL_DWN_FL
      OR      D7961.0  ; NEW_CLAMP_FWD_FL
      ANI     D7814.0  ; UNLOAD  STN     FAULT   RESET
      OUT     D7961.0  ; NEW_CLAMP_FWD_FL
; RUNG NO 224
3231  LD      D7962.1  ; NEW_CLAMP_RET_COMM
      ANI     D7960.0  ; NEW_CLAMP_CYL_UP
      OUT     T167 K100  ; NEW_CLAMP_CYL_UP_FL
; RUNG NO 225
3245  LD      T167  ; NEW_CLAMP_CYL_UP_FL
      OR      D7961.1  ; NEW_CLAMP_RET_FL
      ANI     D7814.0  ; UNLOAD  STN     FAULT   RESET
      OUT     D7961.1  ; NEW_CLAMP_RET_FL
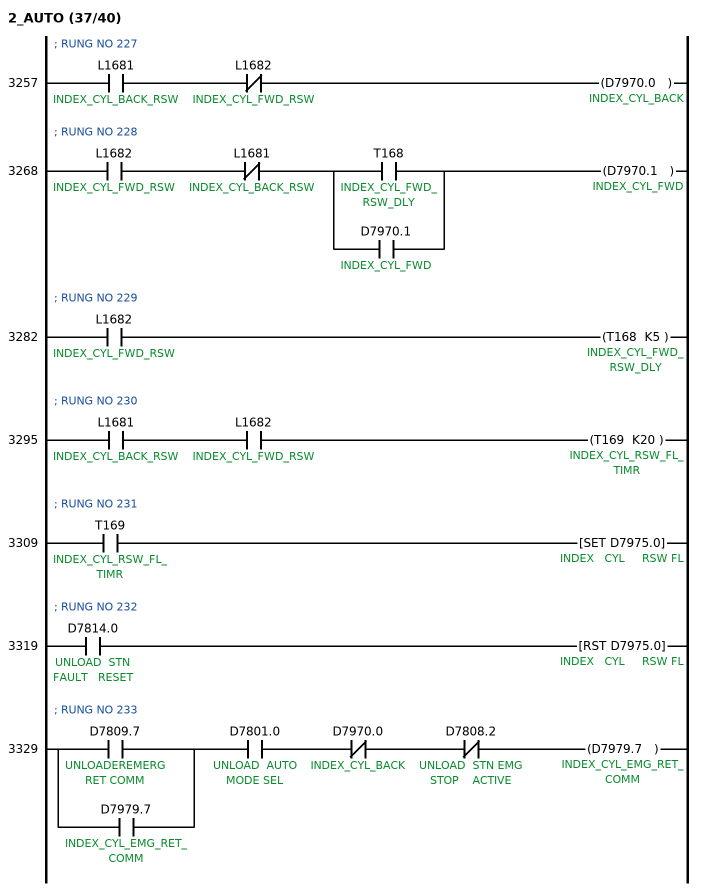
; RUNG NO 227
3257  LD      L1681  ; INDEX_CYL_BACK_RSW
      ANI     L1682  ; INDEX_CYL_FWD_RSW
      OUT     D7970.0  ; INDEX_CYL_BACK
; RUNG NO 228
3268  LD      L1682  ; INDEX_CYL_FWD_RSW
      ANI     L1681  ; INDEX_CYL_BACK_RSW
      LD      T168  ; INDEX_CYL_FWD_RSW_DLY
      OR      D7970.1  ; INDEX_CYL_FWD
      ANB
      OUT     D7970.1  ; INDEX_CYL_FWD
; RUNG NO 229
3282  LD      L1682  ; INDEX_CYL_FWD_RSW
      OUT     T168 K5  ; INDEX_CYL_FWD_RSW_DLY
; RUNG NO 230
3295  LD      L1681  ; INDEX_CYL_BACK_RSW
      AND     L1682  ; INDEX_CYL_FWD_RSW
      OUT     T169 K20  ; INDEX_CYL_RSW_FL_TIMR
; RUNG NO 231
3309  LD      T169  ; INDEX_CYL_RSW_FL_TIMR
      SET     D7975.0  ; INDEX   CYL     RSW FL
; RUNG NO 232
3319  LD      D7814.0  ; UNLOAD  STN     FAULT   RESET
      RST     D7975.0  ; INDEX   CYL     RSW FL
; RUNG NO 233
3329  LD      D7809.7  ; UNLOADEREMERG   RET COMM
      OR      D7979.7  ; INDEX_CYL_EMG_RET_COMM
      AND     D7801.0  ; UNLOAD  AUTO    MODE SEL
      ANI     D7970.0  ; INDEX_CYL_BACK
      ANI     D7808.2  ; UNLOAD  STN EMG STOP    ACTIVE
      OUT     D7979.7  ; INDEX_CYL_EMG_RET_COMM
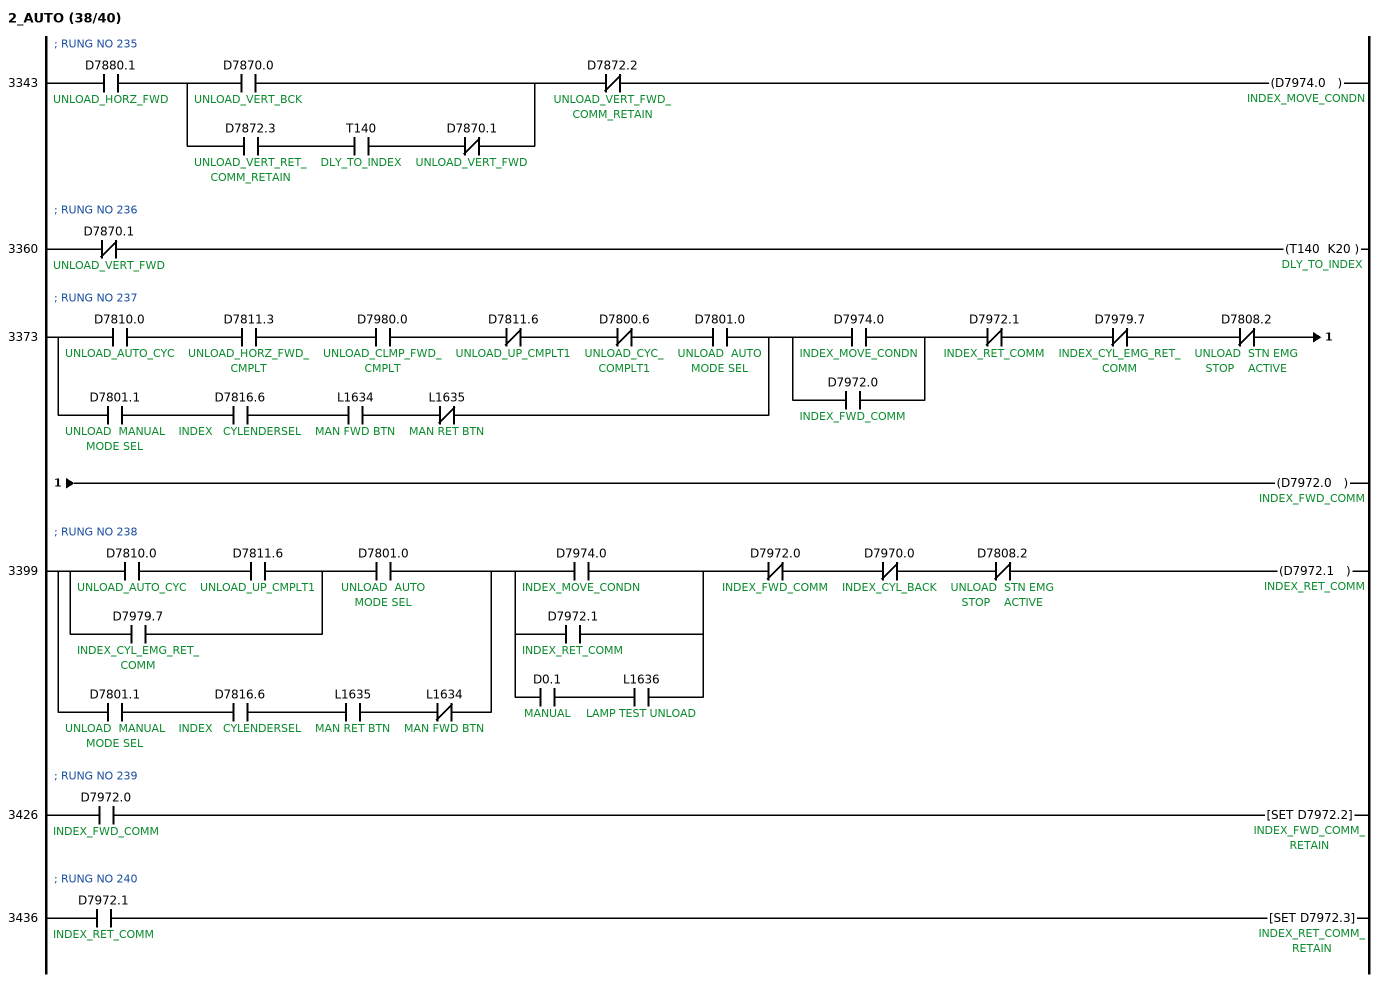
; RUNG NO 235
3343  LD      D7880.1  ; UNLOAD_HORZ_FWD
      LD      D7870.0  ; UNLOAD_VERT_BCK
      LD      D7872.3  ; UNLOAD_VERT_RET_COMM_RETAIN
      AND     T140  ; DLY_TO_INDEX
      ANI     D7870.1  ; UNLOAD_VERT_FWD
      ORB
      ANB
      ANI     D7872.2  ; UNLOAD_VERT_FWD_COMM_RETAIN
      OUT     D7974.0  ; INDEX_MOVE_CONDN
; RUNG NO 236
3360  LDI     D7870.1  ; UNLOAD_VERT_FWD
      OUT     T140 K20  ; DLY_TO_INDEX
; RUNG NO 237
3373  LD      D7810.0  ; UNLOAD_AUTO_CYC
      AND     D7811.3  ; UNLOAD_HORZ_FWD_CMPLT
      AND     D7980.0  ; UNLOAD_CLMP_FWD_CMPLT
      ANI     D7811.6  ; UNLOAD_UP_CMPLT1
      ANI     D7800.6  ; UNLOAD_CYC_COMPLT1
      AND     D7801.0  ; UNLOAD  AUTO    MODE SEL
      LD      D7801.1  ; UNLOAD  MANUAL  MODE SEL
      AND     D7816.6  ; INDEX   CYLENDERSEL
      AND     L1634  ; MAN FWD BTN
      ANI     L1635  ; MAN RET BTN
      ORB
      LD      D7974.0  ; INDEX_MOVE_CONDN
      OR      D7972.0  ; INDEX_FWD_COMM
      ANB
      ANI     D7972.1  ; INDEX_RET_COMM
      ANI     D7979.7  ; INDEX_CYL_EMG_RET_COMM
      ANI     D7808.2  ; UNLOAD  STN EMG STOP    ACTIVE
      OUT     D7972.0  ; INDEX_FWD_COMM
; RUNG NO 238
3399  LD      D7810.0  ; UNLOAD_AUTO_CYC
      AND     D7811.6  ; UNLOAD_UP_CMPLT1
      OR      D7979.7  ; INDEX_CYL_EMG_RET_COMM
      AND     D7801.0  ; UNLOAD  AUTO    MODE SEL
      LD      D7801.1  ; UNLOAD  MANUAL  MODE SEL
      AND     D7816.6  ; INDEX   CYLENDERSEL
      AND     L1635  ; MAN RET BTN
      ANI     L1634  ; MAN FWD BTN
      ORB
      LD      D7974.0  ; INDEX_MOVE_CONDN
      OR      D7972.1  ; INDEX_RET_COMM
      LD      D0.1  ; MANUAL
      AND     L1636  ; LAMP TEST UNLOAD
      ORB
      ANB
      ANI     D7972.0  ; INDEX_FWD_COMM
      ANI     D7970.0  ; INDEX_CYL_BACK
      ANI     D7808.2  ; UNLOAD  STN EMG STOP    ACTIVE
      OUT     D7972.1  ; INDEX_RET_COMM
; RUNG NO 239
3426  LD      D7972.0  ; INDEX_FWD_COMM
      SET     D7972.2  ; INDEX_FWD_COMM_RETAIN
; RUNG NO 240
3436  LD      D7972.1  ; INDEX_RET_COMM
      SET     D7972.3  ; INDEX_RET_COMM_RETAIN
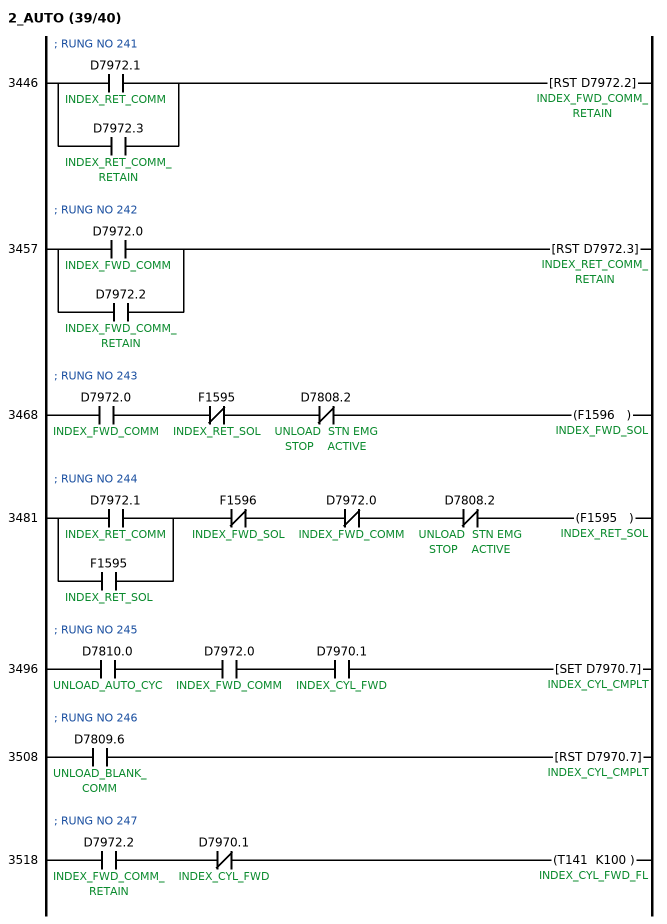
; RUNG NO 241
3446  LD      D7972.1  ; INDEX_RET_COMM
      OR      D7972.3  ; INDEX_RET_COMM_RETAIN
      RST     D7972.2  ; INDEX_FWD_COMM_RETAIN
; RUNG NO 242
3457  LD      D7972.0  ; INDEX_FWD_COMM
      OR      D7972.2  ; INDEX_FWD_COMM_RETAIN
      RST     D7972.3  ; INDEX_RET_COMM_RETAIN
; RUNG NO 243
3468  LD      D7972.0  ; INDEX_FWD_COMM
      ANI     F1595  ; INDEX_RET_SOL
      ANI     D7808.2  ; UNLOAD  STN EMG STOP    ACTIVE
      OUT     F1596  ; INDEX_FWD_SOL
; RUNG NO 244
3481  LD      D7972.1  ; INDEX_RET_COMM
      OR      F1595  ; INDEX_RET_SOL
      ANI     F1596  ; INDEX_FWD_SOL
      ANI     D7972.0  ; INDEX_FWD_COMM
      ANI     D7808.2  ; UNLOAD  STN EMG STOP    ACTIVE
      OUT     F1595  ; INDEX_RET_SOL
; RUNG NO 245
3496  LD      D7810.0  ; UNLOAD_AUTO_CYC
      AND     D7972.0  ; INDEX_FWD_COMM
      AND     D7970.1  ; INDEX_CYL_FWD
      SET     D7970.7  ; INDEX_CYL_CMPLT
; RUNG NO 246
3508  LD      D7809.6  ; UNLOAD_BLANK_COMM
      RST     D7970.7  ; INDEX_CYL_CMPLT
; RUNG NO 247
3518  LD      D7972.2  ; INDEX_FWD_COMM_RETAIN
      ANI     D7970.1  ; INDEX_CYL_FWD
      OUT     T141 K100  ; INDEX_CYL_FWD_FL
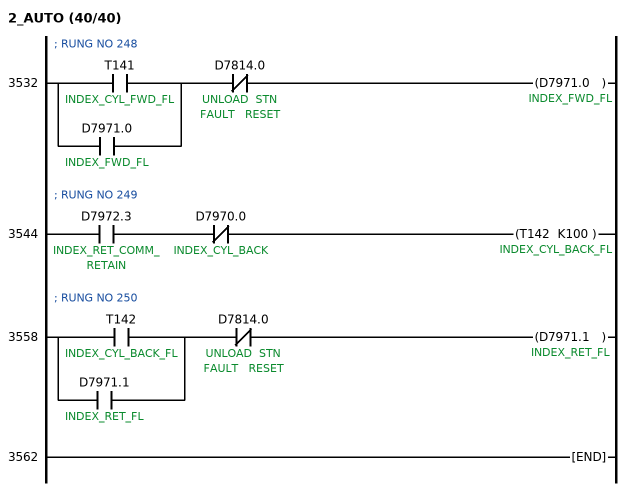
; RUNG NO 248
3532  LD      T141  ; INDEX_CYL_FWD_FL
      OR      D7971.0  ; INDEX_FWD_FL
      ANI     D7814.0  ; UNLOAD  STN     FAULT   RESET
      OUT     D7971.0  ; INDEX_FWD_FL
; RUNG NO 249
3544  LD      D7972.3  ; INDEX_RET_COMM_RETAIN
      ANI     D7970.0  ; INDEX_CYL_BACK
      OUT     T142 K100  ; INDEX_CYL_BACK_FL
; RUNG NO 250
3558  LD      T142  ; INDEX_CYL_BACK_FL
      OR      D7971.1  ; INDEX_RET_FL
      ANI     D7814.0  ; UNLOAD  STN     FAULT   RESET
      OUT     D7971.1  ; INDEX_RET_FL
3562  END
END_PROGRAM

PROGRAM 3_GEN  // CONTROL ALL
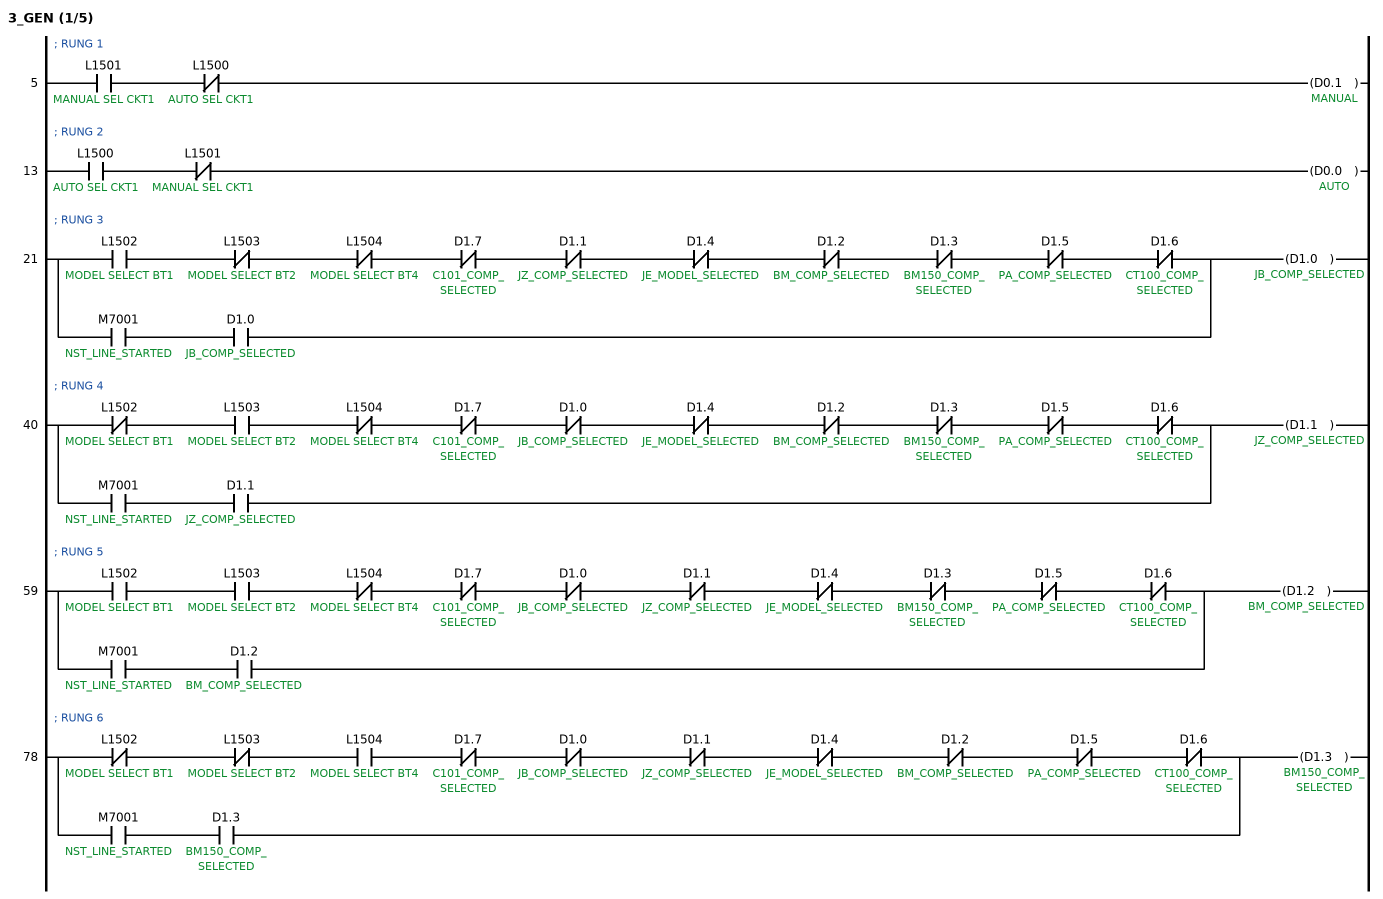
; RUNG 1
5     LD      L1501  ; MANUAL SEL CKT1
      ANI     L1500  ; AUTO SEL CKT1
      OUT     D0.1  ; MANUAL
; RUNG 2
13    LD      L1500  ; AUTO SEL CKT1
      ANI     L1501  ; MANUAL SEL CKT1
      OUT     D0.0  ; AUTO
; RUNG 3
21    LD      L1502  ; MODEL SELECT BT1
      ANI     L1503  ; MODEL SELECT BT2
      ANI     L1504  ; MODEL SELECT BT4
      ANI     D1.7  ; C101_COMP_SELECTED
      ANI     D1.1  ; JZ_COMP_SELECTED
      ANI     D1.4  ; JE_MODEL_SELECTED
      ANI     D1.2  ; BM_COMP_SELECTED
      ANI     D1.3  ; BM150_COMP_SELECTED
      ANI     D1.5  ; PA_COMP_SELECTED
      ANI     D1.6  ; CT100_COMP_SELECTED
      LD      M7001  ; NST_LINE_STARTED
      AND     D1.0  ; JB_COMP_SELECTED
      ORB
      OUT     D1.0  ; JB_COMP_SELECTED
; RUNG 4
40    LDI     L1502  ; MODEL SELECT BT1
      AND     L1503  ; MODEL SELECT BT2
      ANI     L1504  ; MODEL SELECT BT4
      ANI     D1.7  ; C101_COMP_SELECTED
      ANI     D1.0  ; JB_COMP_SELECTED
      ANI     D1.4  ; JE_MODEL_SELECTED
      ANI     D1.2  ; BM_COMP_SELECTED
      ANI     D1.3  ; BM150_COMP_SELECTED
      ANI     D1.5  ; PA_COMP_SELECTED
      ANI     D1.6  ; CT100_COMP_SELECTED
      LD      M7001  ; NST_LINE_STARTED
      AND     D1.1  ; JZ_COMP_SELECTED
      ORB
      OUT     D1.1  ; JZ_COMP_SELECTED
; RUNG 5
59    LD      L1502  ; MODEL SELECT BT1
      AND     L1503  ; MODEL SELECT BT2
      ANI     L1504  ; MODEL SELECT BT4
      ANI     D1.7  ; C101_COMP_SELECTED
      ANI     D1.0  ; JB_COMP_SELECTED
      ANI     D1.1  ; JZ_COMP_SELECTED
      ANI     D1.4  ; JE_MODEL_SELECTED
      ANI     D1.3  ; BM150_COMP_SELECTED
      ANI     D1.5  ; PA_COMP_SELECTED
      ANI     D1.6  ; CT100_COMP_SELECTED
      LD      M7001  ; NST_LINE_STARTED
      AND     D1.2  ; BM_COMP_SELECTED
      ORB
      OUT     D1.2  ; BM_COMP_SELECTED
; RUNG 6
78    LDI     L1502  ; MODEL SELECT BT1
      ANI     L1503  ; MODEL SELECT BT2
      AND     L1504  ; MODEL SELECT BT4
      ANI     D1.7  ; C101_COMP_SELECTED
      ANI     D1.0  ; JB_COMP_SELECTED
      ANI     D1.1  ; JZ_COMP_SELECTED
      ANI     D1.4  ; JE_MODEL_SELECTED
      ANI     D1.2  ; BM_COMP_SELECTED
      ANI     D1.5  ; PA_COMP_SELECTED
      ANI     D1.6  ; CT100_COMP_SELECTED
      LD      M7001  ; NST_LINE_STARTED
      AND     D1.3  ; BM150_COMP_SELECTED
      ORB
      OUT     D1.3  ; BM150_COMP_SELECTED
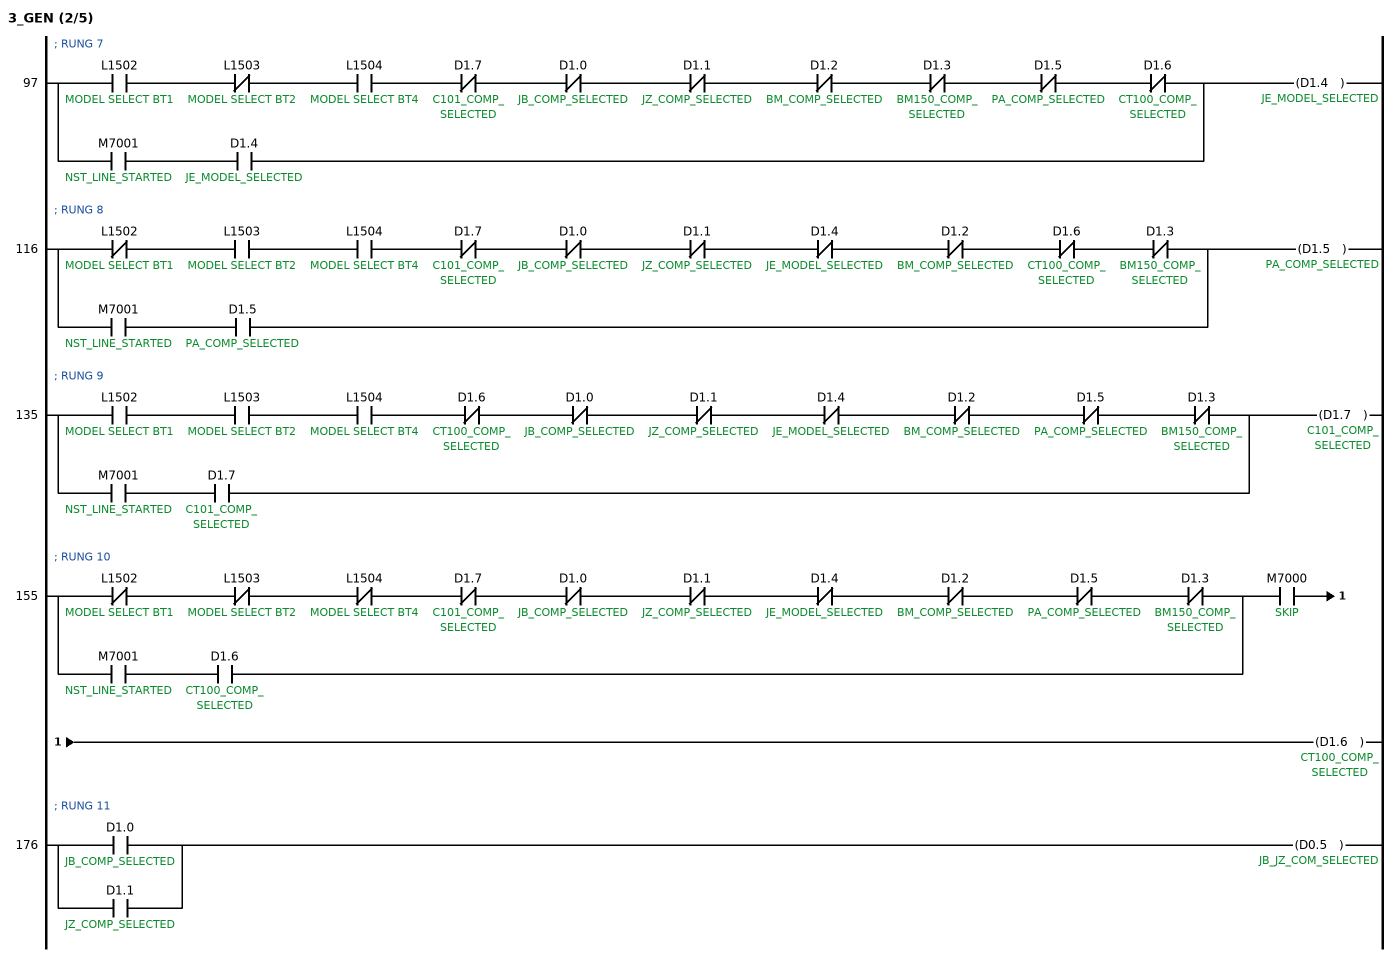
; RUNG 7
97    LD      L1502  ; MODEL SELECT BT1
      ANI     L1503  ; MODEL SELECT BT2
      AND     L1504  ; MODEL SELECT BT4
      ANI     D1.7  ; C101_COMP_SELECTED
      ANI     D1.0  ; JB_COMP_SELECTED
      ANI     D1.1  ; JZ_COMP_SELECTED
      ANI     D1.2  ; BM_COMP_SELECTED
      ANI     D1.3  ; BM150_COMP_SELECTED
      ANI     D1.5  ; PA_COMP_SELECTED
      ANI     D1.6  ; CT100_COMP_SELECTED
      LD      M7001  ; NST_LINE_STARTED
      AND     D1.4  ; JE_MODEL_SELECTED
      ORB
      OUT     D1.4  ; JE_MODEL_SELECTED
; RUNG 8
116   LDI     L1502  ; MODEL SELECT BT1
      AND     L1503  ; MODEL SELECT BT2
      AND     L1504  ; MODEL SELECT BT4
      ANI     D1.7  ; C101_COMP_SELECTED
      ANI     D1.0  ; JB_COMP_SELECTED
      ANI     D1.1  ; JZ_COMP_SELECTED
      ANI     D1.4  ; JE_MODEL_SELECTED
      ANI     D1.2  ; BM_COMP_SELECTED
      ANI     D1.6  ; CT100_COMP_SELECTED
      ANI     D1.3  ; BM150_COMP_SELECTED
      LD      M7001  ; NST_LINE_STARTED
      AND     D1.5  ; PA_COMP_SELECTED
      ORB
      OUT     D1.5  ; PA_COMP_SELECTED
; RUNG 9
135   LD      L1502  ; MODEL SELECT BT1
      AND     L1503  ; MODEL SELECT BT2
      AND     L1504  ; MODEL SELECT BT4
      ANI     D1.6  ; CT100_COMP_SELECTED
      ANI     D1.0  ; JB_COMP_SELECTED
      ANI     D1.1  ; JZ_COMP_SELECTED
      ANI     D1.4  ; JE_MODEL_SELECTED
      ANI     D1.2  ; BM_COMP_SELECTED
      ANI     D1.5  ; PA_COMP_SELECTED
      ANI     D1.3  ; BM150_COMP_SELECTED
      LD      M7001  ; NST_LINE_STARTED
      AND     D1.7  ; C101_COMP_SELECTED
      ORB
      OUT     D1.7  ; C101_COMP_SELECTED
; RUNG 10
155   LDI     L1502  ; MODEL SELECT BT1
      ANI     L1503  ; MODEL SELECT BT2
      ANI     L1504  ; MODEL SELECT BT4
      ANI     D1.7  ; C101_COMP_SELECTED
      ANI     D1.0  ; JB_COMP_SELECTED
      ANI     D1.1  ; JZ_COMP_SELECTED
      ANI     D1.4  ; JE_MODEL_SELECTED
      ANI     D1.2  ; BM_COMP_SELECTED
      ANI     D1.5  ; PA_COMP_SELECTED
      ANI     D1.3  ; BM150_COMP_SELECTED
      LD      M7001  ; NST_LINE_STARTED
      AND     D1.6  ; CT100_COMP_SELECTED
      ORB
      AND     M7000  ; SKIP
      OUT     D1.6  ; CT100_COMP_SELECTED
; RUNG 11
176   LD      D1.0  ; JB_COMP_SELECTED
      OR      D1.1  ; JZ_COMP_SELECTED
      OUT     D0.5  ; JB_JZ_COM_SELECTED
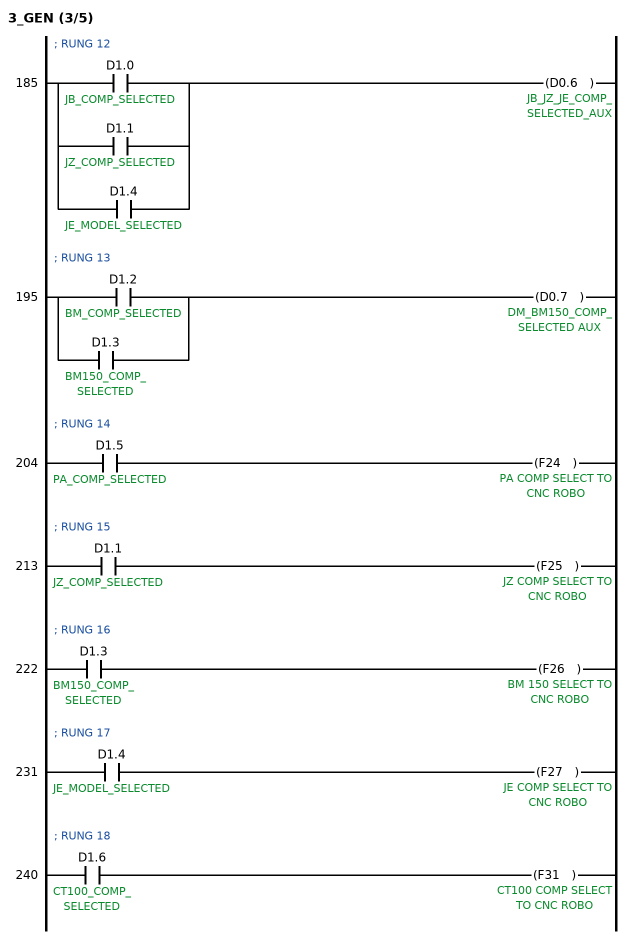
; RUNG 12
185   LD      D1.0  ; JB_COMP_SELECTED
      OR      D1.1  ; JZ_COMP_SELECTED
      OR      D1.4  ; JE_MODEL_SELECTED
      OUT     D0.6  ; JB_JZ_JE_COMP_SELECTED_AUX
; RUNG 13
195   LD      D1.2  ; BM_COMP_SELECTED
      OR      D1.3  ; BM150_COMP_SELECTED
      OUT     D0.7  ; DM_BM150_COMP_SELECTED AUX
; RUNG 14
204   LD      D1.5  ; PA_COMP_SELECTED
      OUT     F24  ; PA COMP SELECT TO CNC ROBO
; RUNG 15
213   LD      D1.1  ; JZ_COMP_SELECTED
      OUT     F25  ; JZ COMP SELECT TO CNC ROBO
; RUNG 16
222   LD      D1.3  ; BM150_COMP_SELECTED
      OUT     F26  ; BM 150 SELECT TO CNC ROBO
; RUNG 17
231   LD      D1.4  ; JE_MODEL_SELECTED
      OUT     F27  ; JE COMP SELECT TO CNC ROBO
; RUNG 18
240   LD      D1.6  ; CT100_COMP_SELECTED
      OUT     F31  ; CT100 COMP SELECT TO CNC ROBO
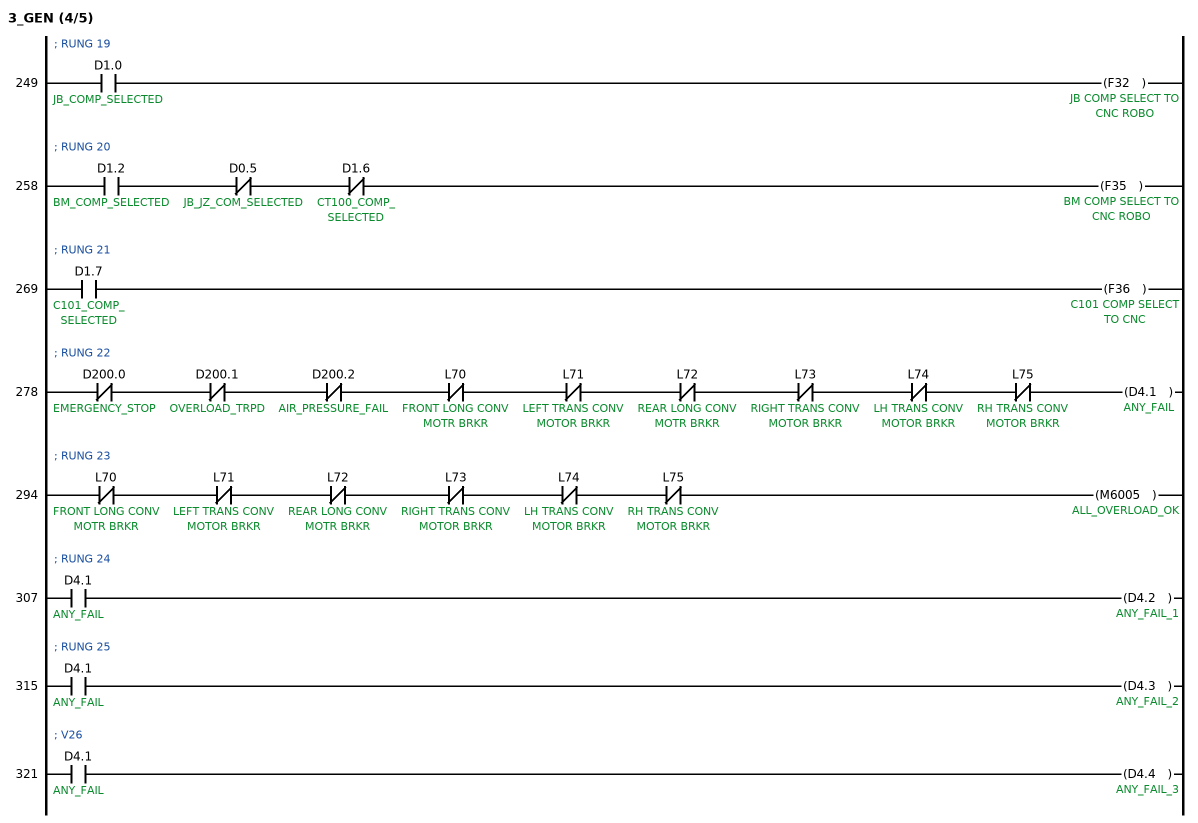
; RUNG 19
249   LD      D1.0  ; JB_COMP_SELECTED
      OUT     F32  ; JB COMP SELECT TO CNC ROBO
; RUNG 20
258   LD      D1.2  ; BM_COMP_SELECTED
      ANI     D0.5  ; JB_JZ_COM_SELECTED
      ANI     D1.6  ; CT100_COMP_SELECTED
      OUT     F35  ; BM COMP SELECT TO CNC ROBO
; RUNG 21
269   LD      D1.7  ; C101_COMP_SELECTED
      OUT     F36  ; C101 COMP SELECT TO CNC
; RUNG 22
278   LDI     D200.0  ; EMERGENCY_STOP
      ANI     D200.1  ; OVERLOAD_TRPD
      ANI     D200.2  ; AIR_PRESSURE_FAIL
      ANI     L70  ; FRONT LONG CONV MOTR BRKR
      ANI     L71  ; LEFT TRANS CONV MOTOR BRKR
      ANI     L72  ; REAR LONG CONV MOTR BRKR
      ANI     L73  ; RIGHT TRANS CONV MOTOR BRKR
      ANI     L74  ; LH TRANS CONV MOTOR BRKR
      ANI     L75  ; RH TRANS CONV MOTOR BRKR
      OUT     D4.1  ; ANY_FAIL
; RUNG 23
294   LDI     L70  ; FRONT LONG CONV MOTR BRKR
      ANI     L71  ; LEFT TRANS CONV MOTOR BRKR
      ANI     L72  ; REAR LONG CONV MOTR BRKR
      ANI     L73  ; RIGHT TRANS CONV MOTOR BRKR
      ANI     L74  ; LH TRANS CONV MOTOR BRKR
      ANI     L75  ; RH TRANS CONV MOTOR BRKR
      OUT     M6005  ; ALL_OVERLOAD_OK
; RUNG 24
307   LD      D4.1  ; ANY_FAIL
      OUT     D4.2  ; ANY_FAIL_1
; RUNG 25
315   LD      D4.1  ; ANY_FAIL
      OUT     D4.3  ; ANY_FAIL_2
; V26
321   LD      D4.1  ; ANY_FAIL
      OUT     D4.4  ; ANY_FAIL_3
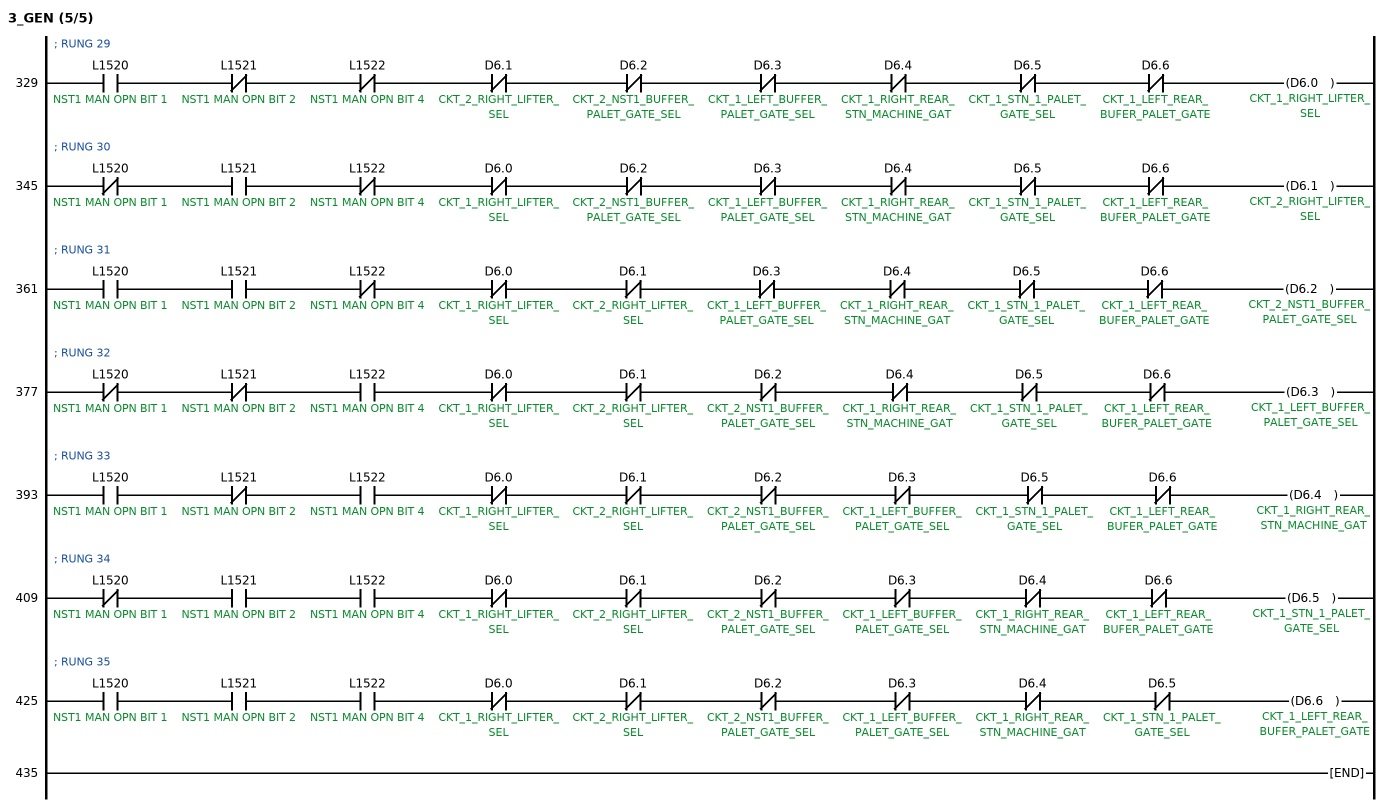
; RUNG 29
329   LD      L1520  ; NST1 MAN OPN BIT 1
      ANI     L1521  ; NST1 MAN OPN BIT 2
      ANI     L1522  ; NST1 MAN OPN BIT 4
      ANI     D6.1  ; CKT_2_RIGHT_LIFTER_SEL
      ANI     D6.2  ; CKT_2_NST1_BUFFER_PALET_GATE_SEL
      ANI     D6.3  ; CKT_1_LEFT_BUFFER_PALET_GATE_SEL
      ANI     D6.4  ; CKT_1_RIGHT_REAR_STN_MACHINE_GAT
      ANI     D6.5  ; CKT_1_STN_1_PALET_GATE_SEL
      ANI     D6.6  ; CKT_1_LEFT_REAR_BUFER_PALET_GATE
      OUT     D6.0  ; CKT_1_RIGHT_LIFTER_SEL
; RUNG 30
345   LDI     L1520  ; NST1 MAN OPN BIT 1
      AND     L1521  ; NST1 MAN OPN BIT 2
      ANI     L1522  ; NST1 MAN OPN BIT 4
      ANI     D6.0  ; CKT_1_RIGHT_LIFTER_SEL
      ANI     D6.2  ; CKT_2_NST1_BUFFER_PALET_GATE_SEL
      ANI     D6.3  ; CKT_1_LEFT_BUFFER_PALET_GATE_SEL
      ANI     D6.4  ; CKT_1_RIGHT_REAR_STN_MACHINE_GAT
      ANI     D6.5  ; CKT_1_STN_1_PALET_GATE_SEL
      ANI     D6.6  ; CKT_1_LEFT_REAR_BUFER_PALET_GATE
      OUT     D6.1  ; CKT_2_RIGHT_LIFTER_SEL
; RUNG 31
361   LD      L1520  ; NST1 MAN OPN BIT 1
      AND     L1521  ; NST1 MAN OPN BIT 2
      ANI     L1522  ; NST1 MAN OPN BIT 4
      ANI     D6.0  ; CKT_1_RIGHT_LIFTER_SEL
      ANI     D6.1  ; CKT_2_RIGHT_LIFTER_SEL
      ANI     D6.3  ; CKT_1_LEFT_BUFFER_PALET_GATE_SEL
      ANI     D6.4  ; CKT_1_RIGHT_REAR_STN_MACHINE_GAT
      ANI     D6.5  ; CKT_1_STN_1_PALET_GATE_SEL
      ANI     D6.6  ; CKT_1_LEFT_REAR_BUFER_PALET_GATE
      OUT     D6.2  ; CKT_2_NST1_BUFFER_PALET_GATE_SEL
; RUNG 32
377   LDI     L1520  ; NST1 MAN OPN BIT 1
      ANI     L1521  ; NST1 MAN OPN BIT 2
      AND     L1522  ; NST1 MAN OPN BIT 4
      ANI     D6.0  ; CKT_1_RIGHT_LIFTER_SEL
      ANI     D6.1  ; CKT_2_RIGHT_LIFTER_SEL
      ANI     D6.2  ; CKT_2_NST1_BUFFER_PALET_GATE_SEL
      ANI     D6.4  ; CKT_1_RIGHT_REAR_STN_MACHINE_GAT
      ANI     D6.5  ; CKT_1_STN_1_PALET_GATE_SEL
      ANI     D6.6  ; CKT_1_LEFT_REAR_BUFER_PALET_GATE
      OUT     D6.3  ; CKT_1_LEFT_BUFFER_PALET_GATE_SEL
; RUNG 33
393   LD      L1520  ; NST1 MAN OPN BIT 1
      ANI     L1521  ; NST1 MAN OPN BIT 2
      AND     L1522  ; NST1 MAN OPN BIT 4
      ANI     D6.0  ; CKT_1_RIGHT_LIFTER_SEL
      ANI     D6.1  ; CKT_2_RIGHT_LIFTER_SEL
      ANI     D6.2  ; CKT_2_NST1_BUFFER_PALET_GATE_SEL
      ANI     D6.3  ; CKT_1_LEFT_BUFFER_PALET_GATE_SEL
      ANI     D6.5  ; CKT_1_STN_1_PALET_GATE_SEL
      ANI     D6.6  ; CKT_1_LEFT_REAR_BUFER_PALET_GATE
      OUT     D6.4  ; CKT_1_RIGHT_REAR_STN_MACHINE_GAT
; RUNG 34
409   LDI     L1520  ; NST1 MAN OPN BIT 1
      AND     L1521  ; NST1 MAN OPN BIT 2
      AND     L1522  ; NST1 MAN OPN BIT 4
      ANI     D6.0  ; CKT_1_RIGHT_LIFTER_SEL
      ANI     D6.1  ; CKT_2_RIGHT_LIFTER_SEL
      ANI     D6.2  ; CKT_2_NST1_BUFFER_PALET_GATE_SEL
      ANI     D6.3  ; CKT_1_LEFT_BUFFER_PALET_GATE_SEL
      ANI     D6.4  ; CKT_1_RIGHT_REAR_STN_MACHINE_GAT
      ANI     D6.6  ; CKT_1_LEFT_REAR_BUFER_PALET_GATE
      OUT     D6.5  ; CKT_1_STN_1_PALET_GATE_SEL
; RUNG 35
425   LD      L1520  ; NST1 MAN OPN BIT 1
      AND     L1521  ; NST1 MAN OPN BIT 2
      AND     L1522  ; NST1 MAN OPN BIT 4
      ANI     D6.0  ; CKT_1_RIGHT_LIFTER_SEL
      ANI     D6.1  ; CKT_2_RIGHT_LIFTER_SEL
      ANI     D6.2  ; CKT_2_NST1_BUFFER_PALET_GATE_SEL
      ANI     D6.3  ; CKT_1_LEFT_BUFFER_PALET_GATE_SEL
      ANI     D6.4  ; CKT_1_RIGHT_REAR_STN_MACHINE_GAT
      ANI     D6.5  ; CKT_1_STN_1_PALET_GATE_SEL
      OUT     D6.6  ; CKT_1_LEFT_REAR_BUFER_PALET_GATE
435   END
END_PROGRAM

PROGRAM 4_LAMPS  // ALL
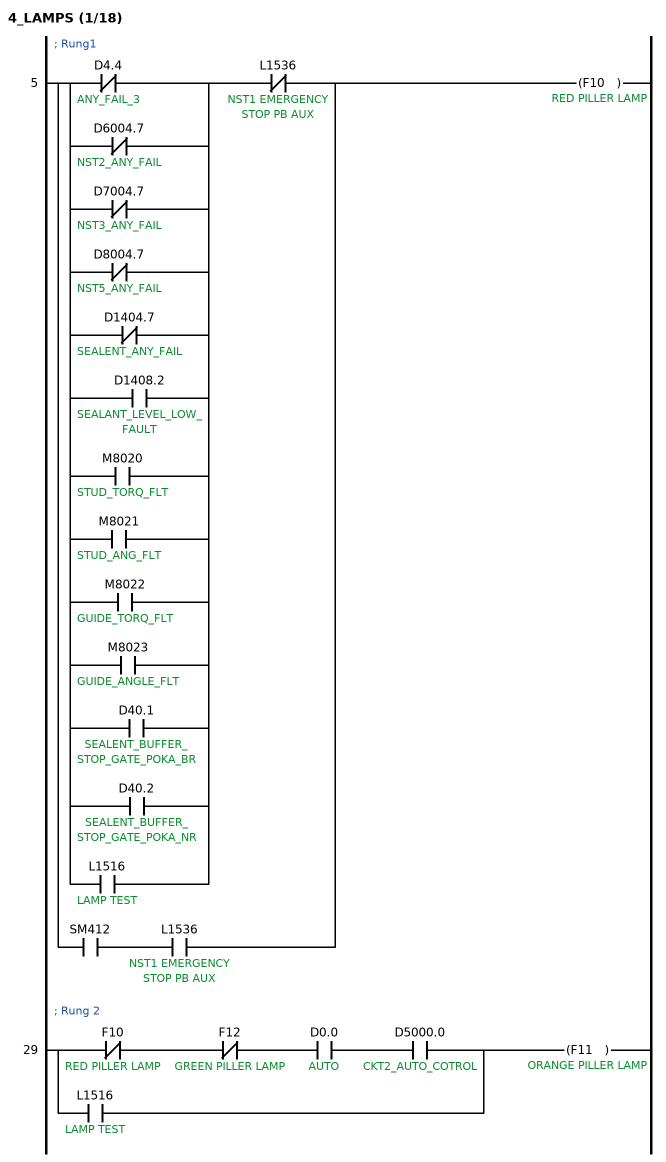
; Rung1
5     LDI     D4.4  ; ANY_FAIL_3
      ORI     D6004.7  ; NST2_ANY_FAIL
      ORI     D7004.7  ; NST3_ANY_FAIL
      ORI     D8004.7  ; NST5_ANY_FAIL
      ORI     D1404.7  ; SEALENT_ANY_FAIL
      OR      D1408.2  ; SEALANT_LEVEL_LOW_FAULT
      OR      M8020  ; STUD_TORQ_FLT
      OR      M8021  ; STUD_ANG_FLT
      OR      M8022  ; GUIDE_TORQ_FLT
      OR      M8023  ; GUIDE_ANGLE_FLT
      OR      D40.1  ; SEALENT_BUFFER_STOP_GATE_POKA_BR
      OR      D40.2  ; SEALENT_BUFFER_STOP_GATE_POKA_NR
      OR      L1516  ; LAMP TEST
      ANI     L1536  ; NST1 EMERGENCY STOP PB AUX
      LD      SM412
      AND     L1536  ; NST1 EMERGENCY STOP PB AUX
      ORB
      OUT     F10  ; RED PILLER LAMP
; Rung 2
29    LDI     F10  ; RED PILLER LAMP
      ANI     F12  ; GREEN PILLER LAMP
      AND     D0.0  ; AUTO
      AND     D5000.0  ; CKT2_AUTO_COTROL
      OR      L1516  ; LAMP TEST
      OUT     F11  ; ORANGE PILLER LAMP
